FUNCTION "FC14 - AUTOMATIC" : VOID	// FC 14
VERSION : 0.1
BEGIN
// (block stored without names or comments; labels and parameter names are numbered)
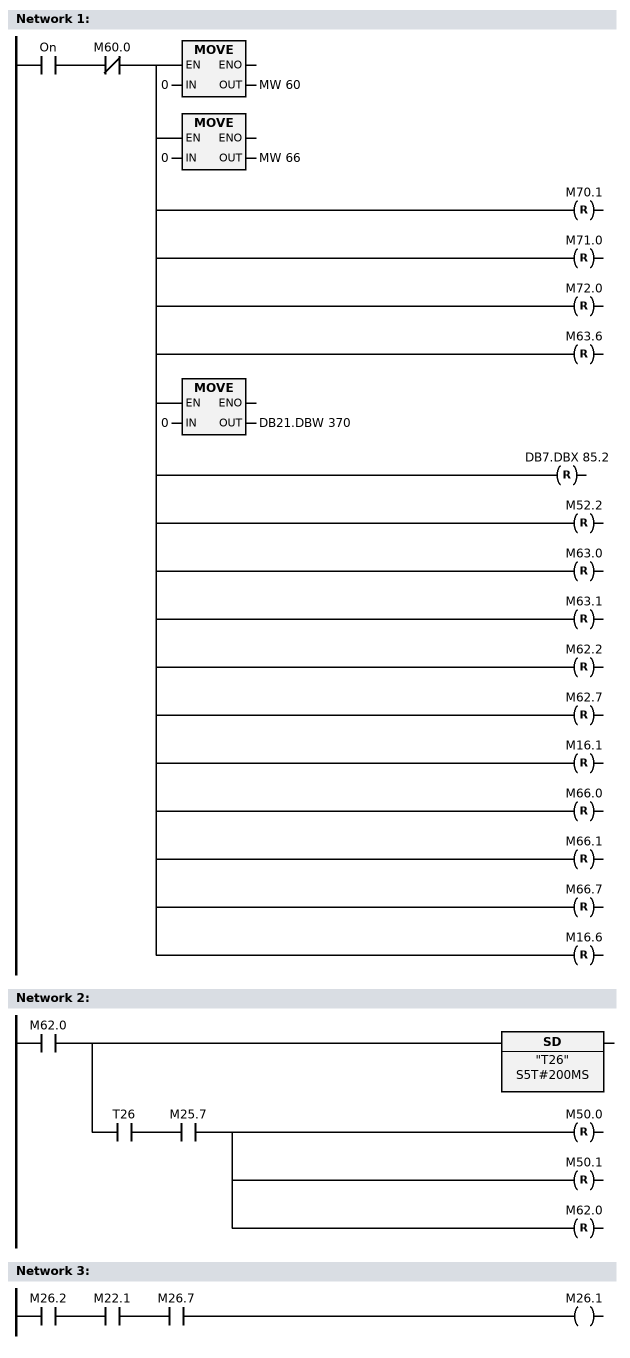
NETWORK
TITLE =
      A     "On";
      AN    "M60.0";
      =     L 24.0;
      A     L 24.0;
      JNB   M001;
      L     0;
      T     MW 60;
M001: NOP   0;
      A     L 24.0;
      JNB   M002;
      L     0;
      T     MW 66;
M002: NOP   0;
      A     L 24.0;
      BLD   102;
      R     "M70.1";
      A     L 24.0;
      BLD   102;
      R     "M71.0";
      A     L 24.0;
      BLD   102;
      R     "M72.0";
      A     L 24.0;
      BLD   102;
      R     "M63.6";
      A     L 24.0;
      JNB   M003;
      L     0;
      T     DB21.DBW 370;
M003: NOP   0;
      A     L 24.0;
      BLD   102;
      R     DB7.DBX 85.2;
      A     L 24.0;
      BLD   102;
      R     "M52.2";
      A     L 24.0;
      BLD   102;
      R     "M63.0";
      A     L 24.0;
      BLD   102;
      R     "M63.1";
      A     L 24.0;
      BLD   102;
      R     "M62.2";
      A     L 24.0;
      BLD   102;
      R     "M62.7";
      A     L 24.0;
      BLD   102;
      R     "M16.1";
      A     L 24.0;
      BLD   102;
      R     "M66.0";
      A     L 24.0;
      BLD   102;
      R     "M66.1";
      A     L 24.0;
      BLD   102;
      R     "M66.7";
      A     L 24.0;
      BLD   102;
      R     "M16.6";
NETWORK
TITLE =
      A     "M62.0";
      =     L 24.0;
      A     L 24.0;
      BLD   102;
      L     S5T#200MS;
      SD    "T26";
      A     L 24.0;
      A     "T26";
      A     "M25.7";
      R     "M50.0";
      R     "M50.1";
      R     "M62.0";
NETWORK
TITLE =
      A     "M26.2";
      A     "M22.1";
      A     "M26.7";
      =     "M26.1";
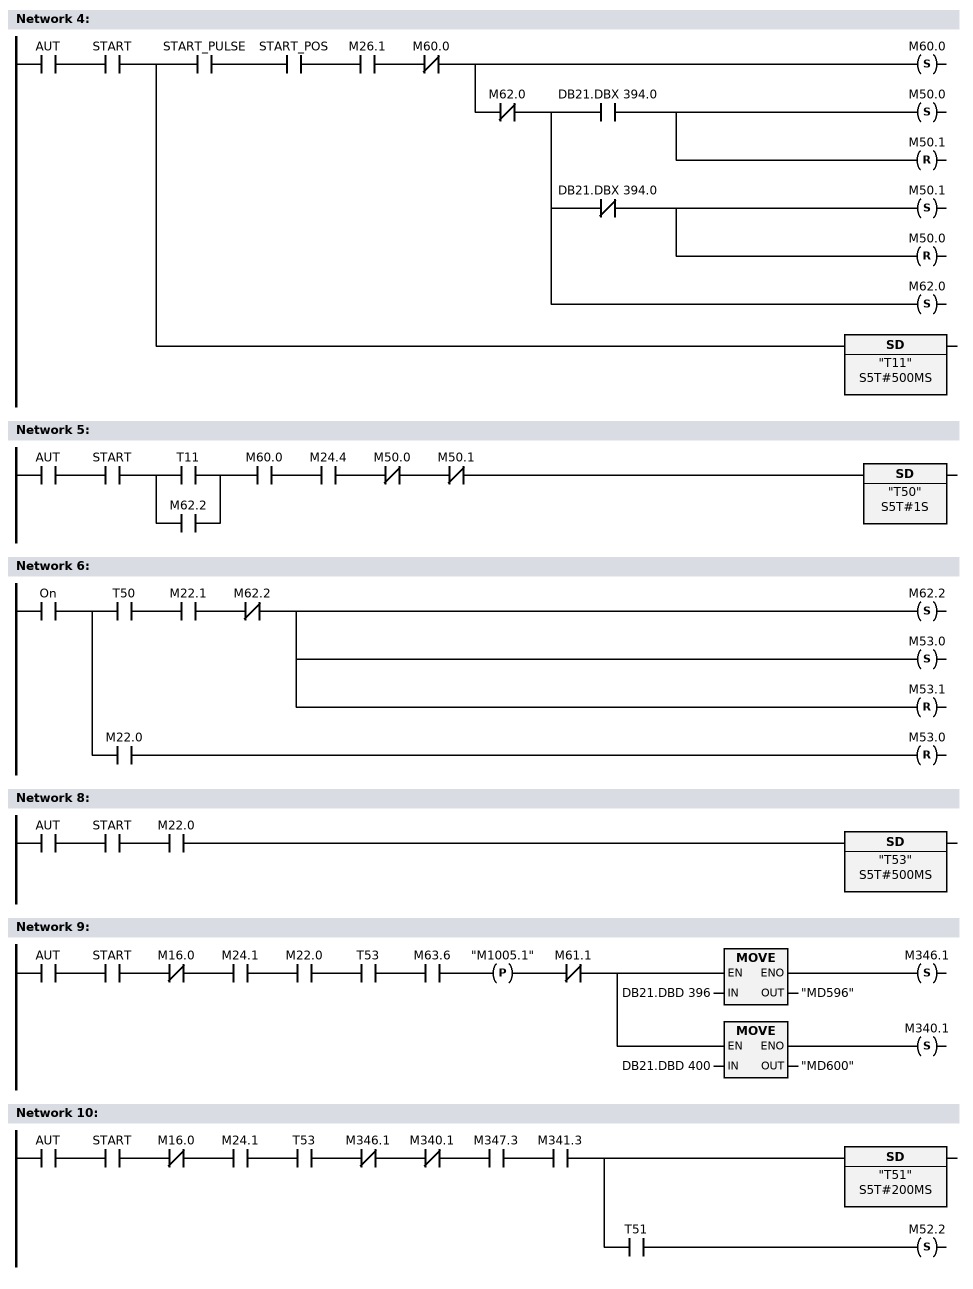
NETWORK
TITLE =
      A     "AUT";
      A     "START";
      =     L 24.0;
      A     L 24.0;
      A     "START_PULSE";
      A     "START_POS";
      A     "M26.1";
      AN    "M60.0";
      =     L 24.1;
      A     L 24.1;
      BLD   102;
      S     "M60.0";
      A     L 24.1;
      AN    "M62.0";
      =     L 24.2;
      A     L 24.2;
      A     DB21.DBX 394.0;
      S     "M50.0";
      R     "M50.1";
      A     L 24.2;
      AN    DB21.DBX 394.0;
      S     "M50.1";
      R     "M50.0";
      A     L 24.2;
      BLD   102;
      S     "M62.0";
      A     L 24.0;
      BLD   102;
      L     S5T#500MS;
      SD    "T11";
NETWORK
TITLE =
      A     "AUT";
      A     "START";
      A(;
      O     "T11";
      O     "M62.2";
      );
      A     "M60.0";
      A     "M24.4";
      AN    "M50.0";
      AN    "M50.1";
      L     S5T#1S;
      SD    "T50";
NETWORK
TITLE =
      A     "On";
      =     L 24.0;
      A     L 24.0;
      A     "T50";
      A     "M22.1";
      AN    "M62.2";
      S     "M62.2";
      S     "M53.0";
      R     "M53.1";
      A     L 24.0;
      A     "M22.0";
      R     "M53.0";
NETWORK
TITLE =
NETWORK
TITLE =
      A     "AUT";
      A     "START";
      A     "M22.0";
      L     S5T#500MS;
      SD    "T53";
NETWORK
TITLE =
      A     "AUT";
      A     "START";
      AN    "M16.0";
      A     "M24.1";
      A     "M22.0";
      A     "T53";
      A     "M63.6";
      FP    "M1005.1";
      AN    "M61.1";
      =     L 24.0;
      A     L 24.0;
      JNB   M004;
      L     DB21.DBD 396;
      T     "MD596";
      SET;
      SAVE;
      CLR;
M004: A     BR;
      S     "M346.1";
      A     L 24.0;
      JNB   M005;
      L     DB21.DBD 400;
      T     "MD600";
      SET;
      SAVE;
      CLR;
M005: A     BR;
      S     "M340.1";
NETWORK
TITLE =
      A     "AUT";
      A     "START";
      AN    "M16.0";
      A     "M24.1";
      A     "T53";
      AN    "M346.1";
      AN    "M340.1";
      A     "M347.3";
      A     "M341.3";
      =     L 24.0;
      A     L 24.0;
      BLD   102;
      L     S5T#200MS;
      SD    "T51";
      A     L 24.0;
      A     "T51";
      S     "M52.2";
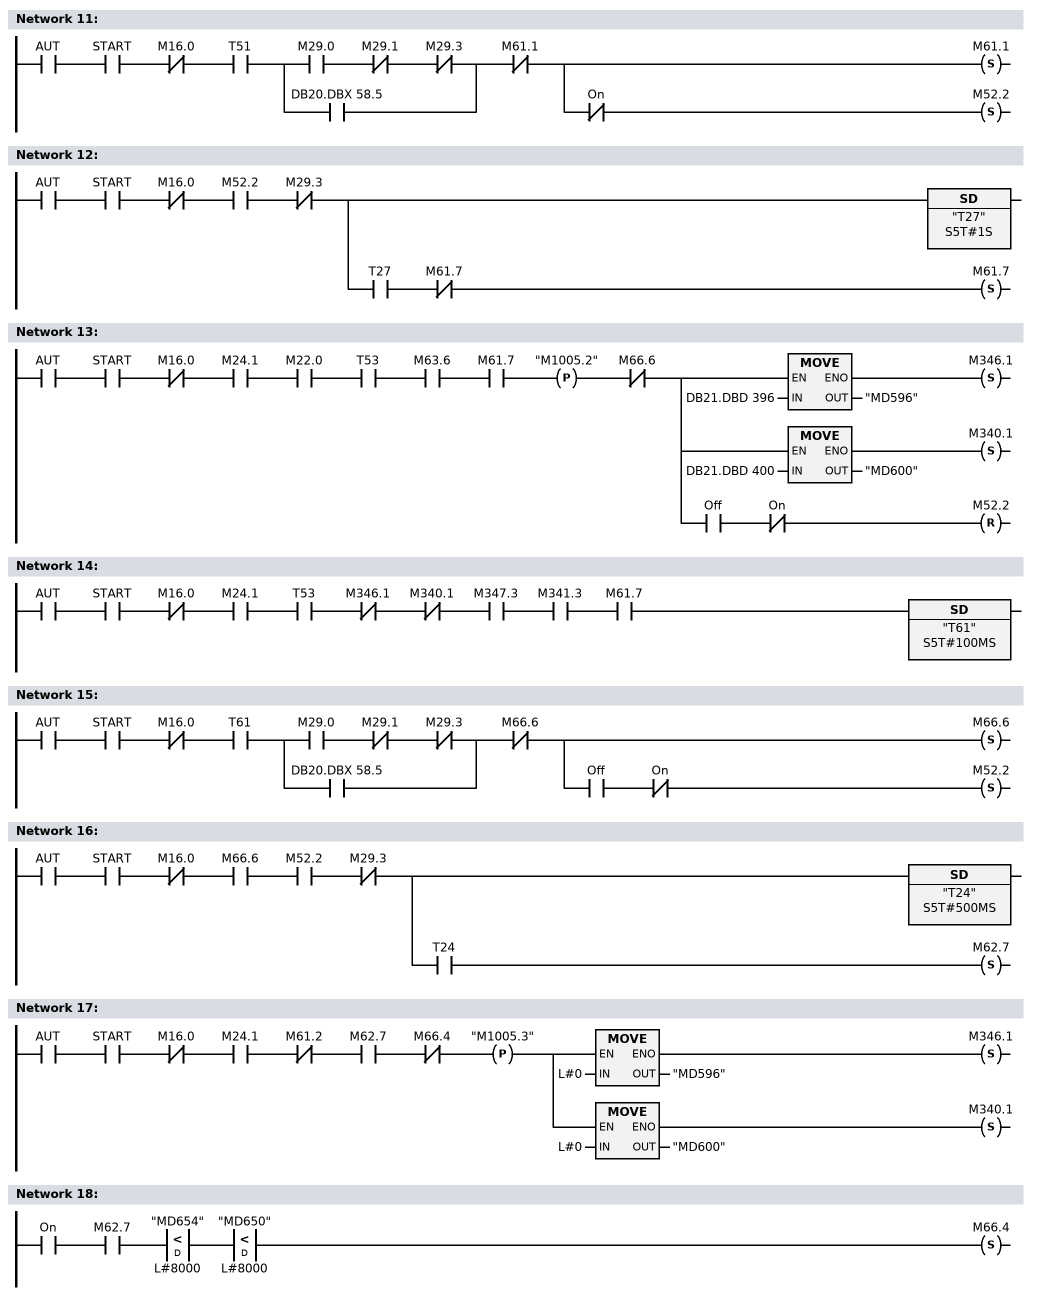
NETWORK
TITLE =
      A     "AUT";
      A     "START";
      AN    "M16.0";
      A     "T51";
      A(;
      A     "M29.0";
      AN    "M29.1";
      AN    "M29.3";
      O     DB20.DBX 58.5;
      );
      AN    "M61.1";
      =     L 24.0;
      A     L 24.0;
      BLD   102;
      S     "M61.1";
      A     L 24.0;
      AN    "On";
      S     "M52.2";
NETWORK
TITLE =
      A     "AUT";
      A     "START";
      AN    "M16.0";
      A     "M52.2";
      AN    "M29.3";
      =     L 24.0;
      A     L 24.0;
      BLD   102;
      L     S5T#1S;
      SD    "T27";
      A     L 24.0;
      A     "T27";
      AN    "M61.7";
      S     "M61.7";
NETWORK
TITLE =
      A     "AUT";
      A     "START";
      AN    "M16.0";
      A     "M24.1";
      A     "M22.0";
      A     "T53";
      A     "M63.6";
      A     "M61.7";
      FP    "M1005.2";
      AN    "M66.6";
      =     L 24.0;
      A     L 24.0;
      JNB   M006;
      L     DB21.DBD 396;
      T     "MD596";
      SET;
      SAVE;
      CLR;
M006: A     BR;
      S     "M346.1";
      A     L 24.0;
      JNB   M007;
      L     DB21.DBD 400;
      T     "MD600";
      SET;
      SAVE;
      CLR;
M007: A     BR;
      S     "M340.1";
      A     L 24.0;
      A     "Off";
      AN    "On";
      R     "M52.2";
NETWORK
TITLE =
      A     "AUT";
      A     "START";
      AN    "M16.0";
      A     "M24.1";
      A     "T53";
      AN    "M346.1";
      AN    "M340.1";
      A     "M347.3";
      A     "M341.3";
      A     "M61.7";
      L     S5T#100MS;
      SD    "T61";
NETWORK
TITLE =
      A     "AUT";
      A     "START";
      AN    "M16.0";
      A     "T61";
      A(;
      A     "M29.0";
      AN    "M29.1";
      AN    "M29.3";
      O     DB20.DBX 58.5;
      );
      AN    "M66.6";
      =     L 24.0;
      A     L 24.0;
      BLD   102;
      S     "M66.6";
      A     L 24.0;
      A     "Off";
      AN    "On";
      S     "M52.2";
NETWORK
TITLE =
      A     "AUT";
      A     "START";
      AN    "M16.0";
      A     "M66.6";
      A     "M52.2";
      AN    "M29.3";
      =     L 24.0;
      A     L 24.0;
      BLD   102;
      L     S5T#500MS;
      SD    "T24";
      A     L 24.0;
      A     "T24";
      S     "M62.7";
NETWORK
TITLE =
      A     "AUT";
      A     "START";
      AN    "M16.0";
      A     "M24.1";
      AN    "M61.2";
      A     "M62.7";
      AN    "M66.4";
      FP    "M1005.3";
      =     L 24.0;
      A     L 24.0;
      JNB   M008;
      L     L#0;
      T     "MD596";
      SET;
      SAVE;
      CLR;
M008: A     BR;
      S     "M346.1";
      A     L 24.0;
      JNB   M009;
      L     L#0;
      T     "MD600";
      SET;
      SAVE;
      CLR;
M009: A     BR;
      S     "M340.1";
NETWORK
TITLE =
      A     "On";
      A     "M62.7";
      A(;
      L     "MD654";
      L     L#8000;
      <D;
      );
      A(;
      L     "MD650";
      L     L#8000;
      <D;
      );
      S     "M66.4";
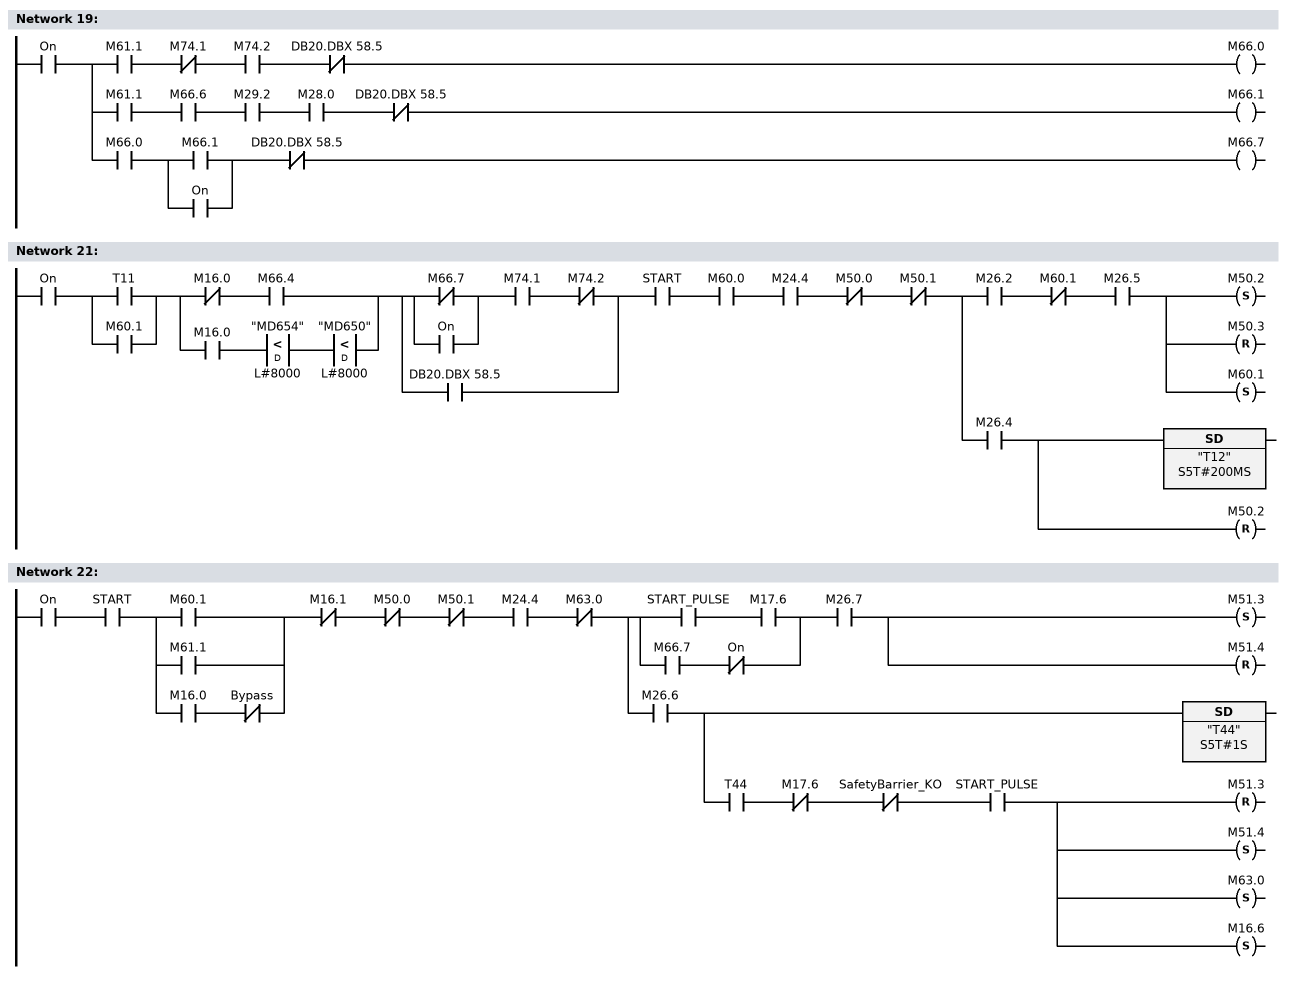
NETWORK
TITLE =
      A     "On";
      =     L 24.0;
      A     L 24.0;
      A     "M61.1";
      AN    "M74.1";
      A     "M74.2";
      AN    DB20.DBX 58.5;
      =     "M66.0";
      A     L 24.0;
      A     "M61.1";
      A     "M66.6";
      A     "M29.2";
      A     "M28.0";
      AN    DB20.DBX 58.5;
      =     "M66.1";
      A     L 24.0;
      A     "M66.0";
      A(;
      O     "M66.1";
      O     "On";
      );
      AN    DB20.DBX 58.5;
      =     "M66.7";
NETWORK
TITLE =
NETWORK
TITLE =
      A     "On";
      A(;
      O     "T11";
      O     "M60.1";
      );
      A(;
      AN    "M16.0";
      A     "M66.4";
      O;
      A     "M16.0";
      A(;
      L     "MD654";
      L     L#8000;
      <D;
      );
      A(;
      L     "MD650";
      L     L#8000;
      <D;
      );
      );
      A(;
      A(;
      ON    "M66.7";
      O     "On";
      );
      A     "M74.1";
      AN    "M74.2";
      O     DB20.DBX 58.5;
      );
      A     "START";
      A     "M60.0";
      A     "M24.4";
      AN    "M50.0";
      AN    "M50.1";
      =     L 24.0;
      A     L 24.0;
      A     "M26.2";
      AN    "M60.1";
      A     "M26.5";
      S     "M50.2";
      R     "M50.3";
      S     "M60.1";
      A     L 24.0;
      A     "M26.4";
      L     S5T#200MS;
      SD    "T12";
      R     "M50.2";
NETWORK
TITLE =
      A     "On";
      A     "START";
      A(;
      O     "M60.1";
      O     "M61.1";
      O;
      A     "M16.0";
      AN    "Bypass";
      );
      AN    "M16.1";
      AN    "M50.0";
      AN    "M50.1";
      A     "M24.4";
      AN    "M63.0";
      =     L 24.0;
      A     L 24.0;
      A(;
      A     "START_PULSE";
      A     "M17.6";
      O;
      A     "M66.7";
      AN    "On";
      );
      A     "M26.7";
      S     "M51.3";
      R     "M51.4";
      A     L 24.0;
      A     "M26.6";
      =     L 24.1;
      A     L 24.1;
      BLD   102;
      L     S5T#1S;
      SD    "T44";
      A     L 24.1;
      A     "T44";
      AN    "M17.6";
      AN    "SafetyBarrier_KO";
      A     "START_PULSE";
      R     "M51.3";
      S     "M51.4";
      S     "M63.0";
      S     "M16.6";
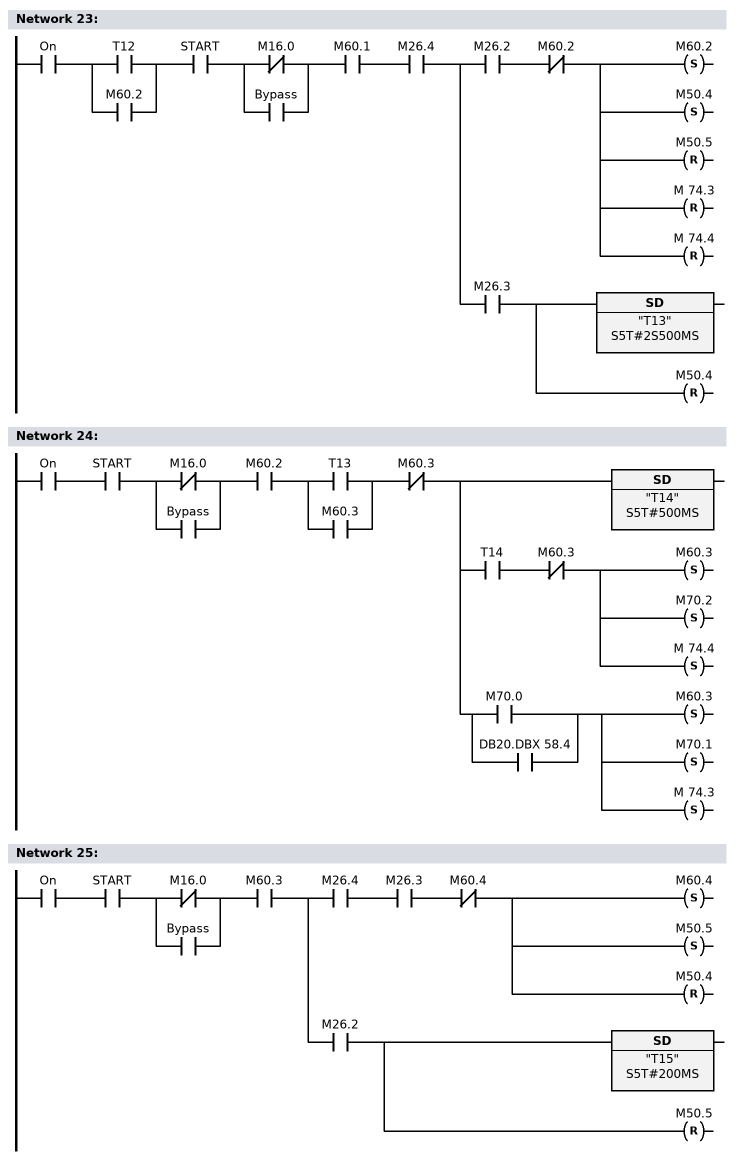
NETWORK
TITLE =
      A     "On";
      A(;
      O     "T12";
      O     "M60.2";
      );
      A     "START";
      A(;
      ON    "M16.0";
      O     "Bypass";
      );
      A     "M60.1";
      A     "M26.4";
      =     L 24.0;
      A     L 24.0;
      A     "M26.2";
      AN    "M60.2";
      S     "M60.2";
      S     "M50.4";
      R     "M50.5";
      R     M 74.3;
      R     M 74.4;
      A     L 24.0;
      A     "M26.3";
      L     S5T#2S500MS;
      SD    "T13";
      R     "M50.4";
NETWORK
TITLE =
      A     "On";
      A     "START";
      A(;
      ON    "M16.0";
      O     "Bypass";
      );
      A     "M60.2";
      A(;
      O     "T13";
      O     "M60.3";
      );
      AN    "M60.3";
      =     L 24.0;
      A     L 24.0;
      BLD   102;
      L     S5T#500MS;
      SD    "T14";
      A     L 24.0;
      A     "T14";
      AN    "M60.3";
      S     "M60.3";
      S     "M70.2";
      S     M 74.4;
      A     L 24.0;
      A(;
      O     "M70.0";
      O     DB20.DBX 58.4;
      );
      S     "M60.3";
      S     "M70.1";
      S     M 74.3;
NETWORK
TITLE =
      A     "On";
      A     "START";
      A(;
      ON    "M16.0";
      O     "Bypass";
      );
      A     "M60.3";
      =     L 24.0;
      A     L 24.0;
      A     "M26.4";
      A     "M26.3";
      AN    "M60.4";
      S     "M60.4";
      S     "M50.5";
      R     "M50.4";
      A     L 24.0;
      A     "M26.2";
      L     S5T#200MS;
      SD    "T15";
      R     "M50.5";
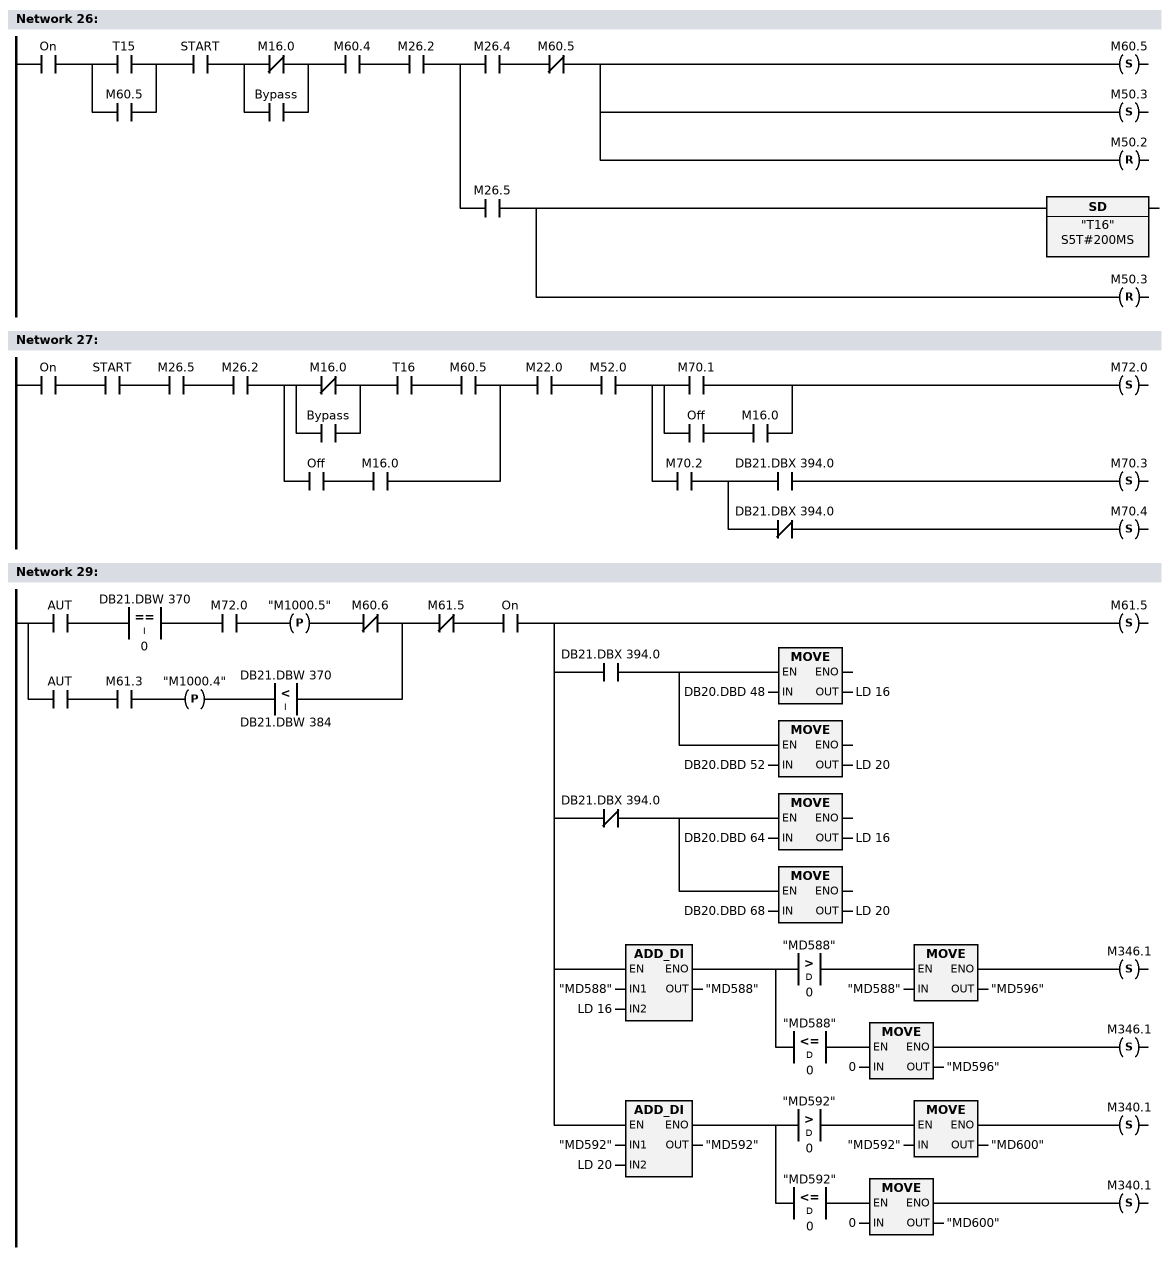
NETWORK
TITLE =
      A     "On";
      A(;
      O     "T15";
      O     "M60.5";
      );
      A     "START";
      A(;
      ON    "M16.0";
      O     "Bypass";
      );
      A     "M60.4";
      A     "M26.2";
      =     L 24.0;
      A     L 24.0;
      A     "M26.4";
      AN    "M60.5";
      S     "M60.5";
      S     "M50.3";
      R     "M50.2";
      A     L 24.0;
      A     "M26.5";
      L     S5T#200MS;
      SD    "T16";
      R     "M50.3";
NETWORK
TITLE =
      A     "On";
      A     "START";
      A     "M26.5";
      A     "M26.2";
      A(;
      A(;
      ON    "M16.0";
      O     "Bypass";
      );
      A     "T16";
      A     "M60.5";
      O;
      A     "Off";
      A     "M16.0";
      );
      A     "M22.0";
      A     "M52.0";
      =     L 24.0;
      A     L 24.0;
      A(;
      O     "M70.1";
      O;
      A     "Off";
      A     "M16.0";
      );
      S     "M72.0";
      A     L 24.0;
      A     "M70.2";
      =     L 24.1;
      A     L 24.1;
      A     DB21.DBX 394.0;
      S     "M70.3";
      A     L 24.1;
      AN    DB21.DBX 394.0;
      S     "M70.4";
NETWORK
TITLE =
NETWORK
TITLE =
      A(;
      A     "AUT";
      A(;
      L     DB21.DBW 370;
      L     0;
      ==I;
      );
      A     "M72.0";
      FP    "M1000.5";
      AN    "M60.6";
      O(;
      A     "AUT";
      A     "M61.3";
      FP    "M1000.4";
      A(;
      L     DB21.DBW 370;
      L     DB21.DBW 384;
      <I;
      );
      );
      );
      AN    "M61.5";
      A     "On";
      =     L 24.0;
      A     L 24.0;
      BLD   102;
      S     "M61.5";
      A     L 24.0;
      A     DB21.DBX 394.0;
      =     L 24.1;
      A     L 24.1;
      JNB   M010;
      L     DB20.DBD 48;
      T     LD 16;
M010: NOP   0;
      A     L 24.1;
      JNB   M011;
      L     DB20.DBD 52;
      T     LD 20;
M011: NOP   0;
      A     L 24.0;
      AN    DB21.DBX 394.0;
      =     L 24.1;
      A     L 24.1;
      JNB   M012;
      L     DB20.DBD 64;
      T     LD 16;
M012: NOP   0;
      A     L 24.1;
      JNB   M013;
      L     DB20.DBD 68;
      T     LD 20;
M013: NOP   0;
      A     L 24.0;
      JNB   M014;
      L     "MD588";
      L     LD 16;
      +D;
      T     "MD588";
      AN    OV;
      SAVE;
      CLR;
M014: A     BR;
      =     L 24.1;
      A     L 24.1;
      A(;
      L     "MD588";
      L     0;
      >D;
      );
      JNB   M015;
      L     "MD588";
      T     "MD596";
      SET;
      SAVE;
      CLR;
M015: A     BR;
      S     "M346.1";
      A     L 24.1;
      A(;
      L     "MD588";
      L     0;
      <=D;
      );
      JNB   M016;
      L     0;
      T     "MD596";
      SET;
      SAVE;
      CLR;
M016: A     BR;
      S     "M346.1";
      A     L 24.0;
      JNB   M017;
      L     "MD592";
      L     LD 20;
      +D;
      T     "MD592";
      AN    OV;
      SAVE;
      CLR;
M017: A     BR;
      =     L 24.1;
      A     L 24.1;
      A(;
      L     "MD592";
      L     0;
      >D;
      );
      JNB   M018;
      L     "MD592";
      T     "MD600";
      SET;
      SAVE;
      CLR;
M018: A     BR;
      S     "M340.1";
      A     L 24.1;
      A(;
      L     "MD592";
      L     0;
      <=D;
      );
      JNB   M019;
      L     0;
      T     "MD600";
      SET;
      SAVE;
      CLR;
M019: A     BR;
      S     "M340.1";
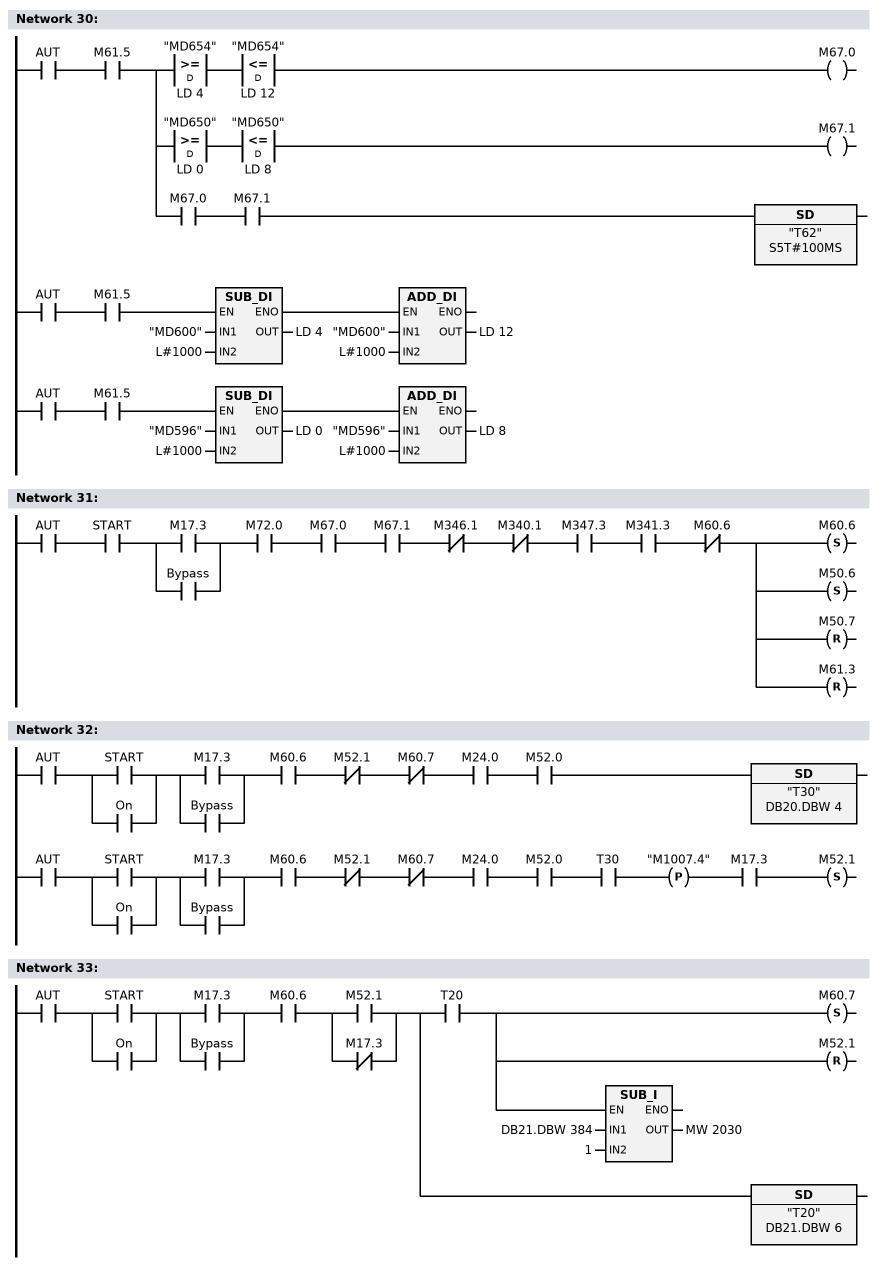
NETWORK
TITLE =
      A     "AUT";
      A     "M61.5";
      =     L 24.0;
      A(;
      A     L 24.0;
      JNB   M020;
      L     "MD600";
      L     L#1000;
      -D;
      T     LD 4;
      AN    OV;
      SAVE;
      CLR;
M020: A     BR;
      );
      JNB   M021;
      L     "MD600";
      L     L#1000;
      +D;
      T     LD 12;
M021: NOP   0;
      A(;
      A     L 24.0;
      JNB   M022;
      L     "MD596";
      L     L#1000;
      -D;
      T     LD 0;
      AN    OV;
      SAVE;
      CLR;
M022: A     BR;
      );
      JNB   M023;
      L     "MD596";
      L     L#1000;
      +D;
      T     LD 8;
M023: NOP   0;
      A     L 24.0;
      A(;
      L     "MD654";
      L     LD 4;
      >=D;
      );
      A(;
      L     "MD654";
      L     LD 12;
      <=D;
      );
      =     "M67.0";
      A     L 24.0;
      A(;
      L     "MD650";
      L     LD 0;
      >=D;
      );
      A(;
      L     "MD650";
      L     LD 8;
      <=D;
      );
      =     "M67.1";
      A     L 24.0;
      A     "M67.0";
      A     "M67.1";
      L     S5T#100MS;
      SD    "T62";
NETWORK
TITLE =
      A     "AUT";
      A     "START";
      A(;
      O     "M17.3";
      O     "Bypass";
      );
      A     "M72.0";
      A     "M67.0";
      A     "M67.1";
      AN    "M346.1";
      AN    "M340.1";
      A     "M347.3";
      A     "M341.3";
      AN    "M60.6";
      S     "M60.6";
      S     "M50.6";
      R     "M50.7";
      R     "M61.3";
NETWORK
TITLE =
      A     "AUT";
      A(;
      O     "START";
      O     "On";
      );
      A(;
      O     "M17.3";
      O     "Bypass";
      );
      A     "M60.6";
      AN    "M52.1";
      AN    "M60.7";
      A     "M24.0";
      A     "M52.0";
      =     L 24.0;
      A     L 24.0;
      BLD   102;
      L     DB20.DBW 4;
      SD    "T30";
      A(;
      A     L 24.0;
      A     "T30";
      FP    "M1007.4";
      );
      A     "M17.3";
      S     "M52.1";
NETWORK
TITLE =
      A     "AUT";
      A(;
      O     "START";
      O     "On";
      );
      A(;
      O     "M17.3";
      O     "Bypass";
      );
      A     "M60.6";
      A(;
      O     "M52.1";
      ON    "M17.3";
      );
      =     L 24.0;
      A     L 24.0;
      A     "T20";
      =     L 24.1;
      A     L 24.1;
      BLD   102;
      S     "M60.7";
      A     L 24.1;
      BLD   102;
      R     "M52.1";
      A     L 24.1;
      JNB   M024;
      L     DB21.DBW 384;
      L     1;
      -I;
      T     MW 2030;
M024: NOP   0;
      A     L 24.0;
      BLD   102;
      L     DB21.DBW 6;
      SD    "T20";
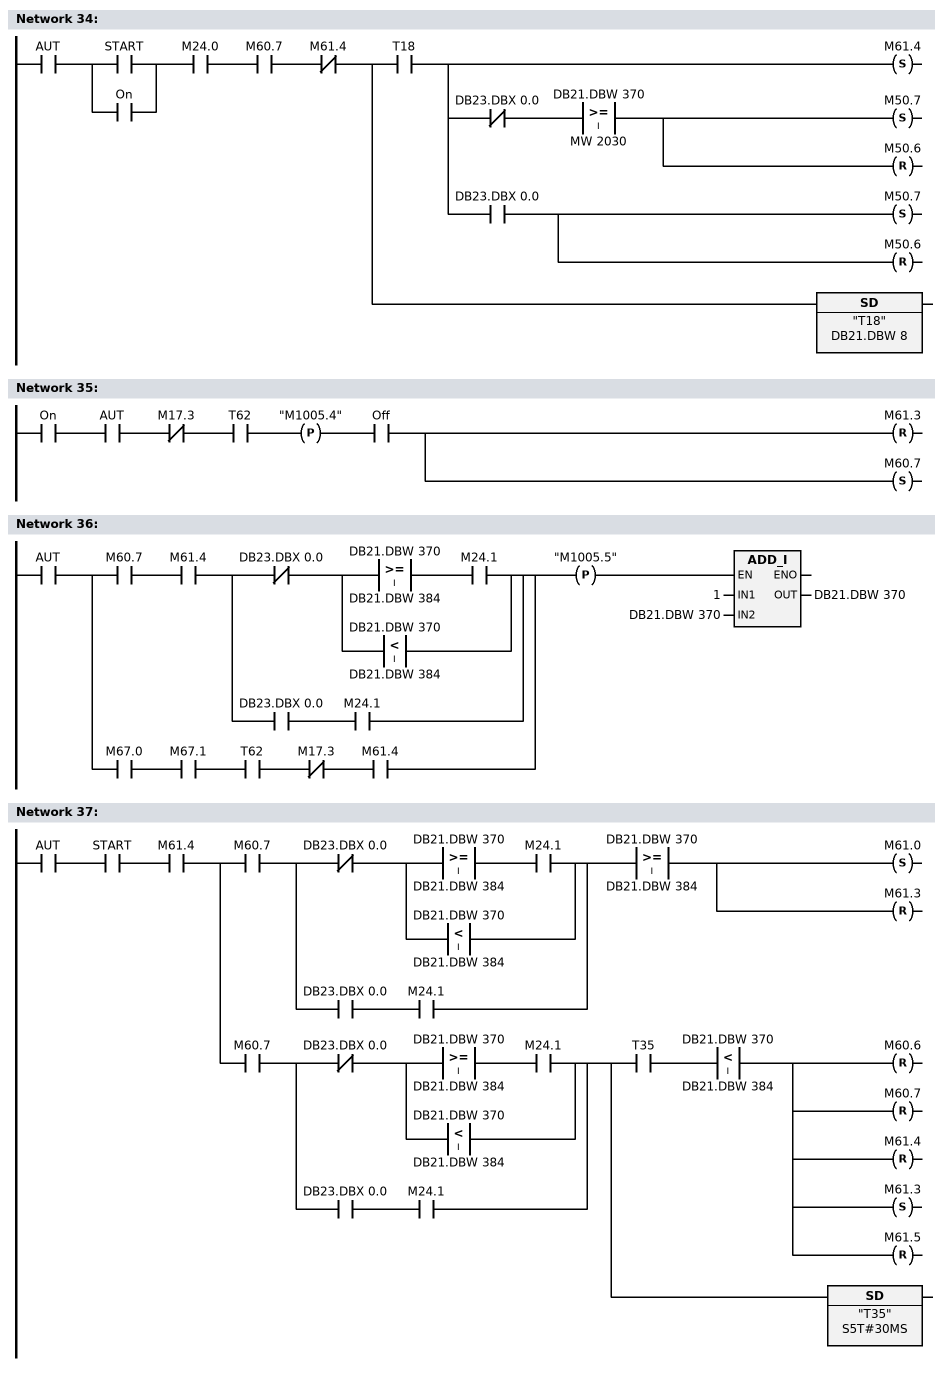
NETWORK
TITLE =
      A     "AUT";
      A(;
      O     "START";
      O     "On";
      );
      A     "M24.0";
      A     "M60.7";
      AN    "M61.4";
      =     L 24.0;
      A     L 24.0;
      A     "T18";
      =     L 24.1;
      A     L 24.1;
      BLD   102;
      S     "M61.4";
      A     L 24.1;
      AN    DB23.DBX 0.0;
      A(;
      L     DB21.DBW 370;
      L     MW 2030;
      >=I;
      );
      S     "M50.7";
      R     "M50.6";
      A     L 24.1;
      A     DB23.DBX 0.0;
      S     "M50.7";
      R     "M50.6";
      A     L 24.0;
      BLD   102;
      L     DB21.DBW 8;
      SD    "T18";
NETWORK
TITLE =
      A     "On";
      A     "AUT";
      AN    "M17.3";
      A     "T62";
      FP    "M1005.4";
      A     "Off";
      R     "M61.3";
      S     "M60.7";
NETWORK
TITLE =
      A     "AUT";
      A(;
      A     "M60.7";
      A     "M61.4";
      A(;
      AN    DB23.DBX 0.0;
      A(;
      A(;
      L     DB21.DBW 370;
      L     DB21.DBW 384;
      >=I;
      );
      A     "M24.1";
      O(;
      L     DB21.DBW 370;
      L     DB21.DBW 384;
      <I;
      );
      );
      O;
      A     DB23.DBX 0.0;
      A     "M24.1";
      );
      O;
      A     "M67.0";
      A     "M67.1";
      A     "T62";
      AN    "M17.3";
      A     "M61.4";
      );
      FP    "M1005.5";
      JNB   M025;
      L     1;
      L     DB21.DBW 370;
      +I;
      T     DB21.DBW 370;
M025: NOP   0;
NETWORK
TITLE =
      A     "AUT";
      A     "START";
      A     "M61.4";
      =     L 24.0;
      A     L 24.0;
      A     "M60.7";
      A(;
      AN    DB23.DBX 0.0;
      A(;
      A(;
      L     DB21.DBW 370;
      L     DB21.DBW 384;
      >=I;
      );
      A     "M24.1";
      O(;
      L     DB21.DBW 370;
      L     DB21.DBW 384;
      <I;
      );
      );
      O;
      A     DB23.DBX 0.0;
      A     "M24.1";
      );
      A(;
      L     DB21.DBW 370;
      L     DB21.DBW 384;
      >=I;
      );
      S     "M61.0";
      R     "M61.3";
      A     L 24.0;
      A     "M60.7";
      A(;
      AN    DB23.DBX 0.0;
      A(;
      A(;
      L     DB21.DBW 370;
      L     DB21.DBW 384;
      >=I;
      );
      A     "M24.1";
      O(;
      L     DB21.DBW 370;
      L     DB21.DBW 384;
      <I;
      );
      );
      O;
      A     DB23.DBX 0.0;
      A     "M24.1";
      );
      =     L 24.1;
      A     L 24.1;
      A     "T35";
      A(;
      L     DB21.DBW 370;
      L     DB21.DBW 384;
      <I;
      );
      R     "M60.6";
      R     "M60.7";
      R     "M61.4";
      S     "M61.3";
      R     "M61.5";
      A     L 24.1;
      BLD   102;
      L     S5T#30MS;
      SD    "T35";
NETWORK
TITLE =
NETWORK
TITLE =
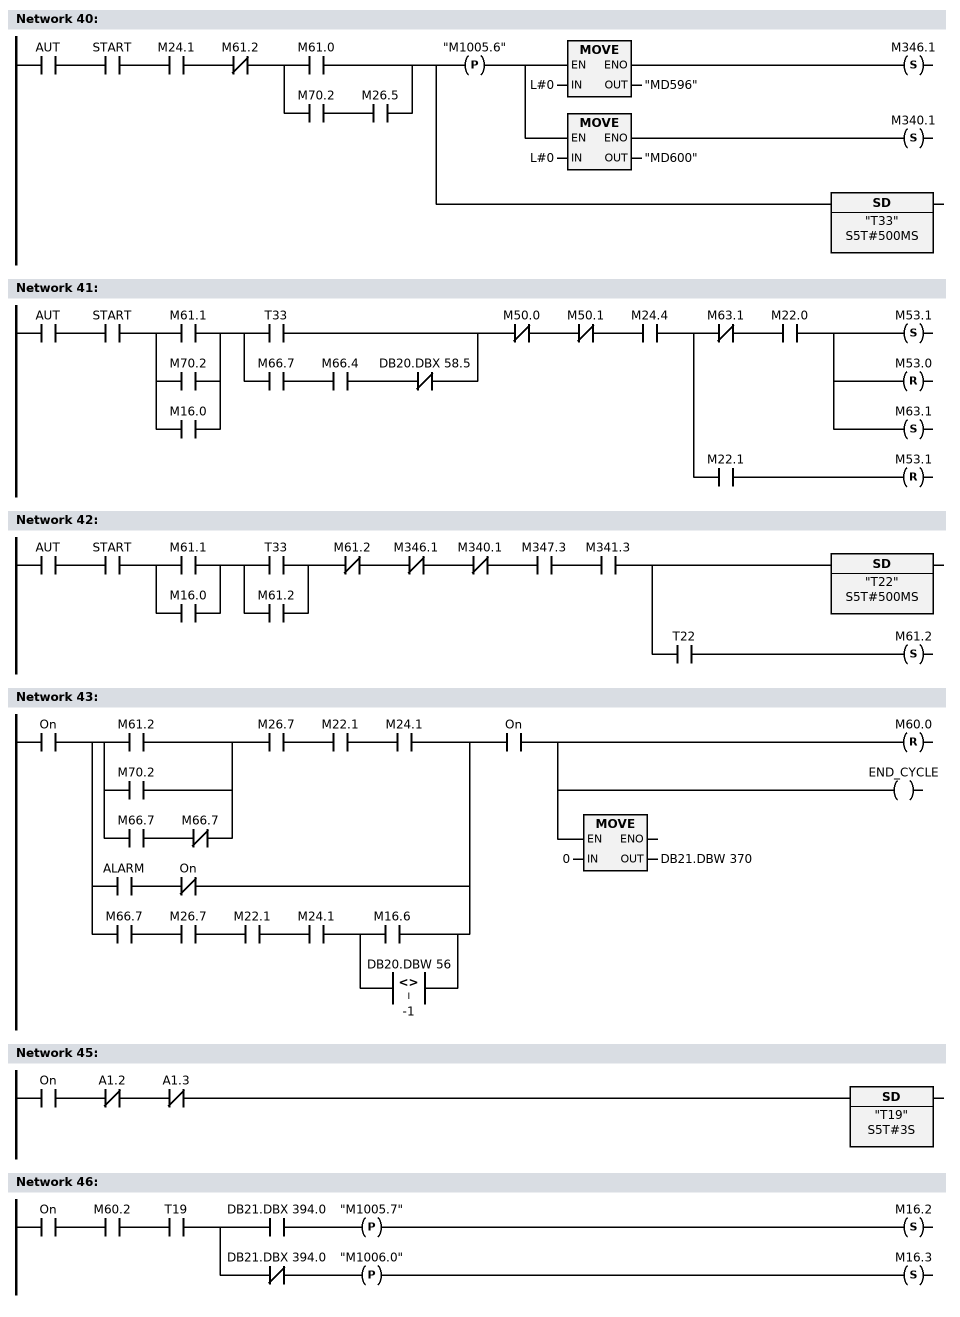
NETWORK
TITLE =
      A     "AUT";
      A     "START";
      A     "M24.1";
      AN    "M61.2";
      A(;
      O     "M61.0";
      O;
      A     "M70.2";
      A     "M26.5";
      );
      =     L 24.0;
      A     L 24.0;
      FP    "M1005.6";
      =     L 24.1;
      A     L 24.1;
      JNB   M026;
      L     L#0;
      T     "MD596";
      SET;
      SAVE;
      CLR;
M026: A     BR;
      S     "M346.1";
      A     L 24.1;
      JNB   M027;
      L     L#0;
      T     "MD600";
      SET;
      SAVE;
      CLR;
M027: A     BR;
      S     "M340.1";
      A     L 24.0;
      BLD   102;
      L     S5T#500MS;
      SD    "T33";
NETWORK
TITLE =
      A     "AUT";
      A     "START";
      A(;
      O     "M61.1";
      O     "M70.2";
      O     "M16.0";
      );
      A(;
      O     "T33";
      O;
      A     "M66.7";
      A     "M66.4";
      AN    DB20.DBX 58.5;
      );
      AN    "M50.0";
      AN    "M50.1";
      A     "M24.4";
      =     L 24.0;
      A     L 24.0;
      AN    "M63.1";
      A     "M22.0";
      S     "M53.1";
      R     "M53.0";
      S     "M63.1";
      A     L 24.0;
      A     "M22.1";
      R     "M53.1";
NETWORK
TITLE =
      A     "AUT";
      A     "START";
      A(;
      O     "M61.1";
      O     "M16.0";
      );
      A(;
      O     "T33";
      O     "M61.2";
      );
      AN    "M61.2";
      AN    "M346.1";
      AN    "M340.1";
      A     "M347.3";
      A     "M341.3";
      =     L 24.0;
      A     L 24.0;
      BLD   102;
      L     S5T#500MS;
      SD    "T22";
      A     L 24.0;
      A     "T22";
      S     "M61.2";
NETWORK
TITLE =
      A     "On";
      A(;
      A(;
      O     "M61.2";
      O     "M70.2";
      O;
      A     "M66.7";
      AN    "M66.7";
      );
      A     "M26.7";
      A     "M22.1";
      A     "M24.1";
      O;
      A     "ALARM";
      AN    "On";
      O;
      A     "M66.7";
      A     "M26.7";
      A     "M22.1";
      A     "M24.1";
      A(;
      O     "M16.6";
      O(;
      L     DB20.DBW 56;
      L     -1;
      <>I;
      );
      );
      );
      A     "On";
      =     L 24.0;
      A     L 24.0;
      BLD   102;
      R     "M60.0";
      A     L 24.0;
      BLD   102;
      =     "END_CYCLE";
      A     L 24.0;
      JNB   M028;
      L     0;
      T     DB21.DBW 370;
M028: NOP   0;
NETWORK
TITLE =
NETWORK
TITLE =
      A     "On";
      AN    "A1.2";
      AN    "A1.3";
      L     S5T#3S;
      SD    "T19";
NETWORK
TITLE =
      A     "On";
      A     "M60.2";
      A     "T19";
      =     L 24.0;
      A     L 24.0;
      A     DB21.DBX 394.0;
      FP    "M1005.7";
      S     "M16.2";
      A     L 24.0;
      AN    DB21.DBX 394.0;
      FP    "M1006.0";
      S     "M16.3";
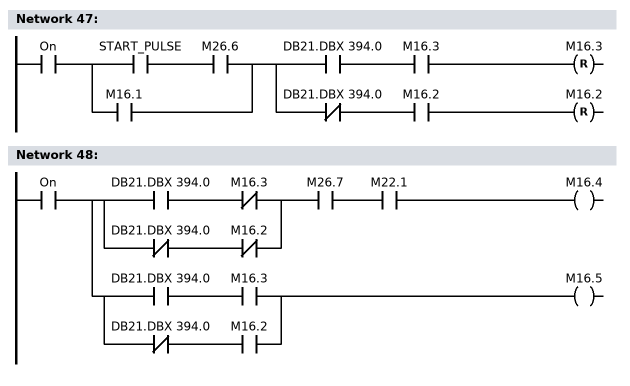
NETWORK
TITLE =
      A     "On";
      A(;
      A     "START_PULSE";
      A     "M26.6";
      O     "M16.1";
      );
      =     L 24.0;
      A     L 24.0;
      A     DB21.DBX 394.0;
      A     "M16.3";
      R     "M16.3";
      A     L 24.0;
      AN    DB21.DBX 394.0;
      A     "M16.2";
      R     "M16.2";
NETWORK
TITLE =
      A     "On";
      =     L 24.0;
      A     L 24.0;
      A(;
      A     DB21.DBX 394.0;
      AN    "M16.3";
      O;
      AN    DB21.DBX 394.0;
      AN    "M16.2";
      );
      A     "M26.7";
      A     "M22.1";
      =     "M16.4";
      A     L 24.0;
      A(;
      A     DB21.DBX 394.0;
      A     "M16.3";
      O;
      AN    DB21.DBX 394.0;
      A     "M16.2";
      );
      =     "M16.5";
END_FUNCTION

FUNCTION "FC16 - ALARMS" : VOID	// FC 16
VERSION : 0.1
BEGIN
// (block stored without names or comments; labels and parameter names are numbered)
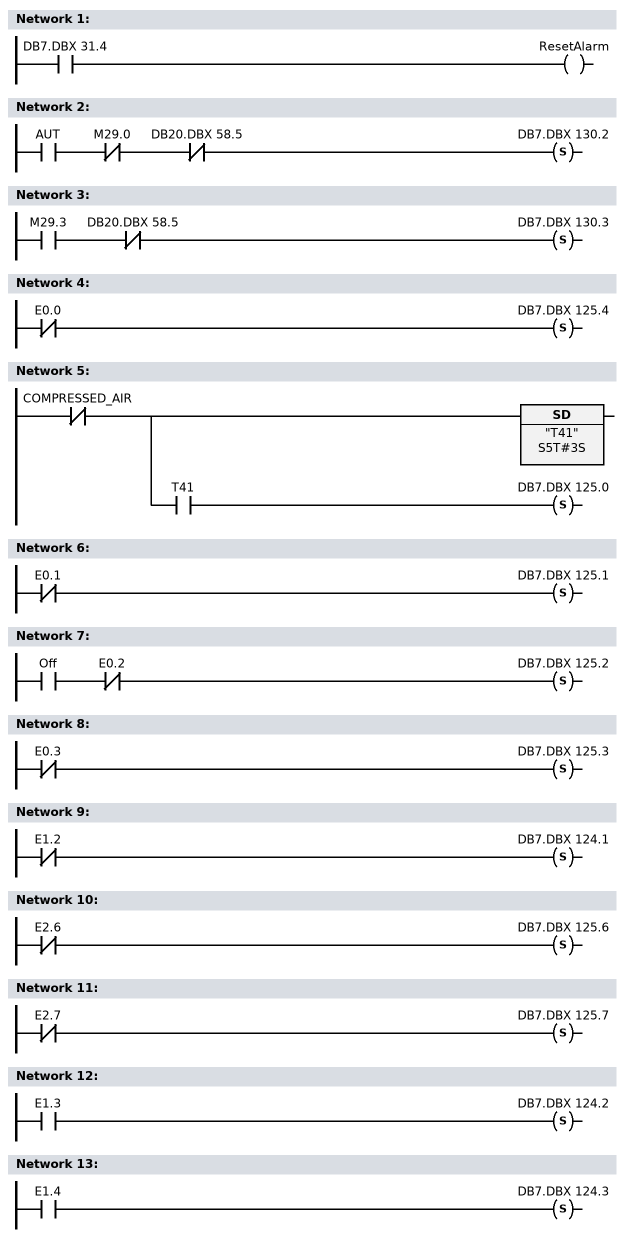
NETWORK
TITLE =
      A     DB7.DBX 31.4;
      =     "ResetAlarm";
NETWORK
TITLE =
      A     "AUT";
      AN    "M29.0";
      AN    DB20.DBX 58.5;
      S     DB7.DBX 130.2;
NETWORK
TITLE =
      A     "M29.3";
      AN    DB20.DBX 58.5;
      S     DB7.DBX 130.3;
NETWORK
TITLE =
      AN    "E0.0";
      S     DB7.DBX 125.4;
NETWORK
TITLE =
      AN    "COMPRESSED_AIR";
      =     L 1.0;
      A     L 1.0;
      BLD   102;
      L     S5T#3S;
      SD    "T41";
      A     L 1.0;
      A     "T41";
      S     DB7.DBX 125.0;
NETWORK
TITLE =
      AN    "E0.1";
      S     DB7.DBX 125.1;
NETWORK
TITLE =
      A     "Off";
      AN    "E0.2";
      S     DB7.DBX 125.2;
NETWORK
TITLE =
      AN    "E0.3";
      S     DB7.DBX 125.3;
NETWORK
TITLE =
      AN    "E1.2";
      S     DB7.DBX 124.1;
NETWORK
TITLE =
      AN    "E2.6";
      S     DB7.DBX 125.6;
NETWORK
TITLE =
      AN    "E2.7";
      S     DB7.DBX 125.7;
NETWORK
TITLE =
      A     "E1.3";
      S     DB7.DBX 124.2;
NETWORK
TITLE =
      A     "E1.4";
      S     DB7.DBX 124.3;
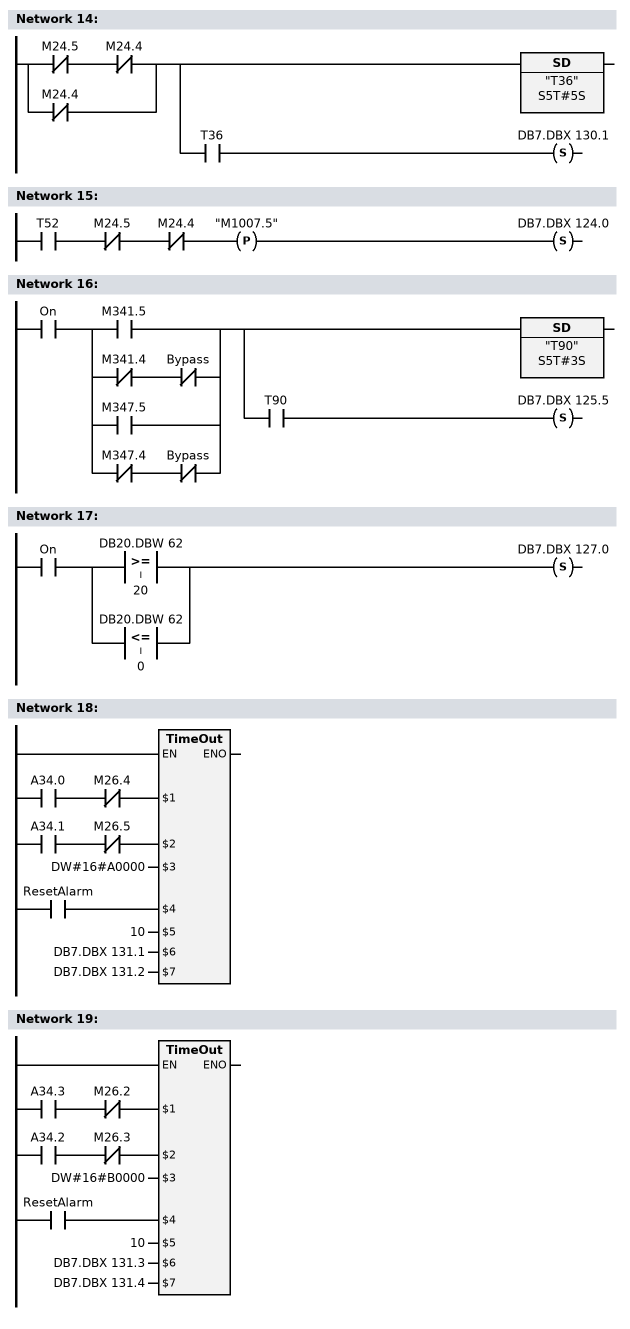
NETWORK
TITLE =
      AN    "M24.5";
      AN    "M24.4";
      ON    "M24.4";
      =     L 1.0;
      A     L 1.0;
      BLD   102;
      L     S5T#5S;
      SD    "T36";
      A     L 1.0;
      A     "T36";
      S     DB7.DBX 130.1;
NETWORK
TITLE =
      A     "T52";
      AN    "M24.5";
      AN    "M24.4";
      FP    "M1007.5";
      S     DB7.DBX 124.0;
NETWORK
TITLE =
      A     "On";
      A(;
      O     "M341.5";
      O;
      AN    "M341.4";
      AN    "Bypass";
      O     "M347.5";
      O;
      AN    "M347.4";
      AN    "Bypass";
      );
      =     L 1.0;
      A     L 1.0;
      BLD   102;
      L     S5T#3S;
      SD    "T90";
      A     L 1.0;
      A     "T90";
      S     DB7.DBX 125.5;
NETWORK
TITLE =
      A     "On";
      A(;
      O(;
      L     DB20.DBW 62;
      L     20;
      >=I;
      );
      O(;
      L     DB20.DBW 62;
      L     0;
      <=I;
      );
      );
      S     DB7.DBX 127.0;
NETWORK
TITLE =
      A     "A34.0";
      AN    "M26.4";
      =     L 1.0;
      BLD   103;
      A     "A34.1";
      AN    "M26.5";
      =     L 1.1;
      BLD   103;
      A     "ResetAlarm";
      =     L 1.2;
      BLD   103;
      CALL  "TimeOut" (
           $1                       := L 1.0,
           $2                       := L 1.1,
           $3                       := DW#16#A0000,
           $4                       := L 1.2,
           $5                       := 10,
           $6                       := DB7.DBX 131.1,
           $7                       := DB7.DBX 131.2);
      NOP   0;
NETWORK
TITLE =
      A     "A34.3";
      AN    "M26.2";
      =     L 1.0;
      BLD   103;
      A     "A34.2";
      AN    "M26.3";
      =     L 1.1;
      BLD   103;
      A     "ResetAlarm";
      =     L 1.2;
      BLD   103;
      CALL  "TimeOut" (
           $1                       := L 1.0,
           $2                       := L 1.1,
           $3                       := DW#16#B0000,
           $4                       := L 1.2,
           $5                       := 10,
           $6                       := DB7.DBX 131.3,
           $7                       := DB7.DBX 131.4);
      NOP   0;
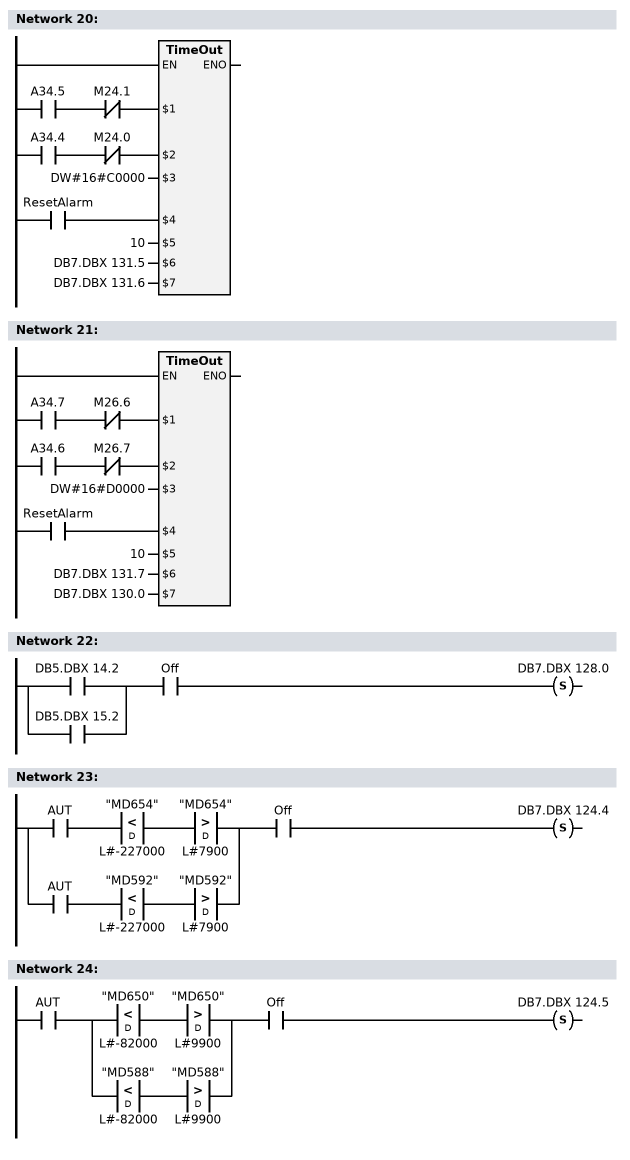
NETWORK
TITLE =
      A     "A34.5";
      AN    "M24.1";
      =     L 1.0;
      BLD   103;
      A     "A34.4";
      AN    "M24.0";
      =     L 1.1;
      BLD   103;
      A     "ResetAlarm";
      =     L 1.2;
      BLD   103;
      CALL  "TimeOut" (
           $1                       := L 1.0,
           $2                       := L 1.1,
           $3                       := DW#16#C0000,
           $4                       := L 1.2,
           $5                       := 10,
           $6                       := DB7.DBX 131.5,
           $7                       := DB7.DBX 131.6);
      NOP   0;
NETWORK
TITLE =
      A     "A34.7";
      AN    "M26.6";
      =     L 1.0;
      BLD   103;
      A     "A34.6";
      AN    "M26.7";
      =     L 1.1;
      BLD   103;
      A     "ResetAlarm";
      =     L 1.2;
      BLD   103;
      CALL  "TimeOut" (
           $1                       := L 1.0,
           $2                       := L 1.1,
           $3                       := DW#16#D0000,
           $4                       := L 1.2,
           $5                       := 10,
           $6                       := DB7.DBX 131.7,
           $7                       := DB7.DBX 130.0);
      NOP   0;
NETWORK
TITLE =
      A(;
      O     DB5.DBX 14.2;
      O     DB5.DBX 15.2;
      );
      A     "Off";
      S     DB7.DBX 128.0;
NETWORK
TITLE =
      A(;
      A     "AUT";
      A(;
      L     "MD654";
      L     L#-227000;
      <D;
      );
      A(;
      L     "MD654";
      L     L#7900;
      >D;
      );
      O;
      A     "AUT";
      A(;
      L     "MD592";
      L     L#-227000;
      <D;
      );
      A(;
      L     "MD592";
      L     L#7900;
      >D;
      );
      );
      A     "Off";
      S     DB7.DBX 124.4;
NETWORK
TITLE =
      A     "AUT";
      A(;
      A(;
      L     "MD650";
      L     L#-82000;
      <D;
      );
      A(;
      L     "MD650";
      L     L#9900;
      >D;
      );
      O;
      A(;
      L     "MD588";
      L     L#-82000;
      <D;
      );
      A(;
      L     "MD588";
      L     L#9900;
      >D;
      );
      );
      A     "Off";
      S     DB7.DBX 124.5;
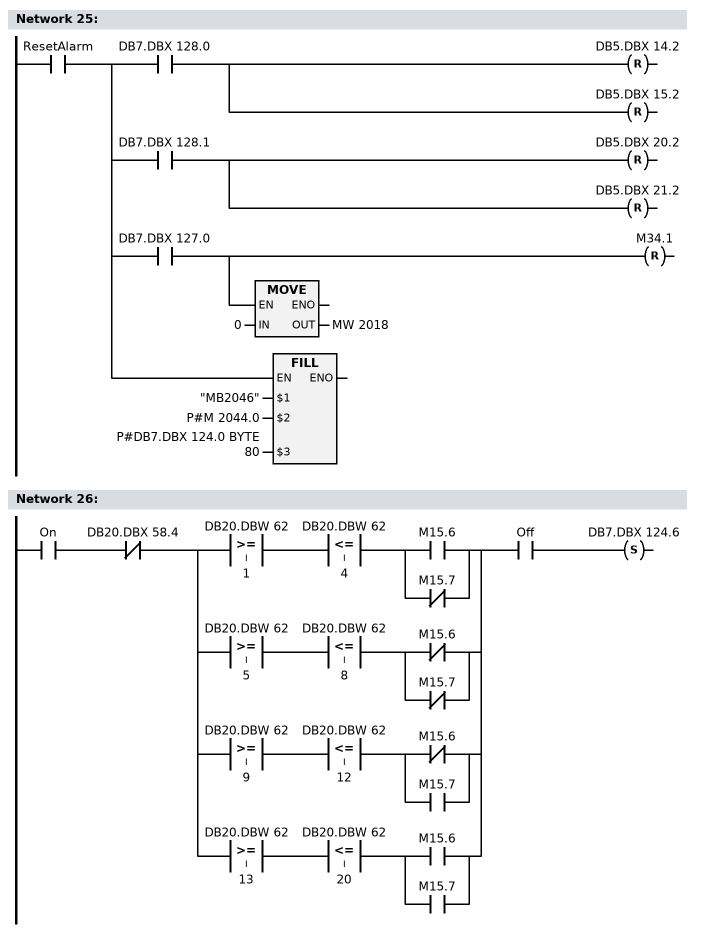
NETWORK
TITLE =
      A     "ResetAlarm";
      =     L 1.0;
      A     L 1.0;
      A     DB7.DBX 128.0;
      R     DB5.DBX 14.2;
      R     DB5.DBX 15.2;
      A     L 1.0;
      A     DB7.DBX 128.1;
      R     DB5.DBX 20.2;
      R     DB5.DBX 21.2;
      A     L 1.0;
      A     DB7.DBX 127.0;
      =     L 1.1;
      A     L 1.1;
      BLD   102;
      R     "M34.1";
      A     L 1.1;
      JNB   M001;
      L     0;
      T     MW 2018;
M001: NOP   0;
      A     L 1.0;
      JNB   M002;
      CALL  "FILL" (
           $1                       := "MB2046",
           $2                       := P#M 2044.0,
           $3                       := P#DB7.DBX 124.0 BYTE 80);
M002: NOP   0;
NETWORK
TITLE =
      A     "On";
      AN    DB20.DBX 58.4;
      A(;
      A(;
      L     DB20.DBW 62;
      L     1;
      >=I;
      );
      A(;
      L     DB20.DBW 62;
      L     4;
      <=I;
      );
      A(;
      O     "M15.6";
      ON    "M15.7";
      );
      O;
      A(;
      L     DB20.DBW 62;
      L     5;
      >=I;
      );
      A(;
      L     DB20.DBW 62;
      L     8;
      <=I;
      );
      A(;
      ON    "M15.6";
      ON    "M15.7";
      );
      O;
      A(;
      L     DB20.DBW 62;
      L     9;
      >=I;
      );
      A(;
      L     DB20.DBW 62;
      L     12;
      <=I;
      );
      A(;
      ON    "M15.6";
      O     "M15.7";
      );
      O;
      A(;
      L     DB20.DBW 62;
      L     13;
      >=I;
      );
      A(;
      L     DB20.DBW 62;
      L     20;
      <=I;
      );
      A(;
      O     "M15.6";
      O     "M15.7";
      );
      );
      A     "Off";
      S     DB7.DBX 124.6;
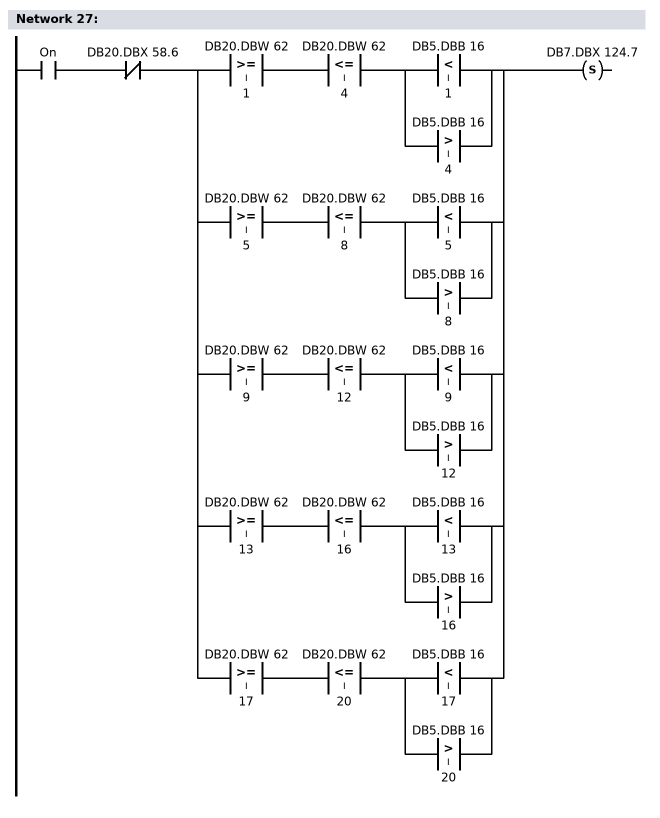
NETWORK
TITLE =
      A     "On";
      AN    DB20.DBX 58.6;
      A(;
      A(;
      L     DB20.DBW 62;
      L     1;
      >=I;
      );
      A(;
      L     DB20.DBW 62;
      L     4;
      <=I;
      );
      A(;
      O(;
      L     DB5.DBB 16;
      L     1;
      <I;
      );
      O(;
      L     DB5.DBB 16;
      L     4;
      >I;
      );
      );
      O;
      A(;
      L     DB20.DBW 62;
      L     5;
      >=I;
      );
      A(;
      L     DB20.DBW 62;
      L     8;
      <=I;
      );
      A(;
      O(;
      L     DB5.DBB 16;
      L     5;
      <I;
      );
      O(;
      L     DB5.DBB 16;
      L     8;
      >I;
      );
      );
      O;
      A(;
      L     DB20.DBW 62;
      L     9;
      >=I;
      );
      A(;
      L     DB20.DBW 62;
      L     12;
      <=I;
      );
      A(;
      O(;
      L     DB5.DBB 16;
      L     9;
      <I;
      );
      O(;
      L     DB5.DBB 16;
      L     12;
      >I;
      );
      );
      O;
      A(;
      L     DB20.DBW 62;
      L     13;
      >=I;
      );
      A(;
      L     DB20.DBW 62;
      L     16;
      <=I;
      );
      A(;
      O(;
      L     DB5.DBB 16;
      L     13;
      <I;
      );
      O(;
      L     DB5.DBB 16;
      L     16;
      >I;
      );
      );
      O;
      A(;
      L     DB20.DBW 62;
      L     17;
      >=I;
      );
      A(;
      L     DB20.DBW 62;
      L     20;
      <=I;
      );
      A(;
      O(;
      L     DB5.DBB 16;
      L     17;
      <I;
      );
      O(;
      L     DB5.DBB 16;
      L     20;
      >I;
      );
      );
      );
      S     DB7.DBX 124.7;
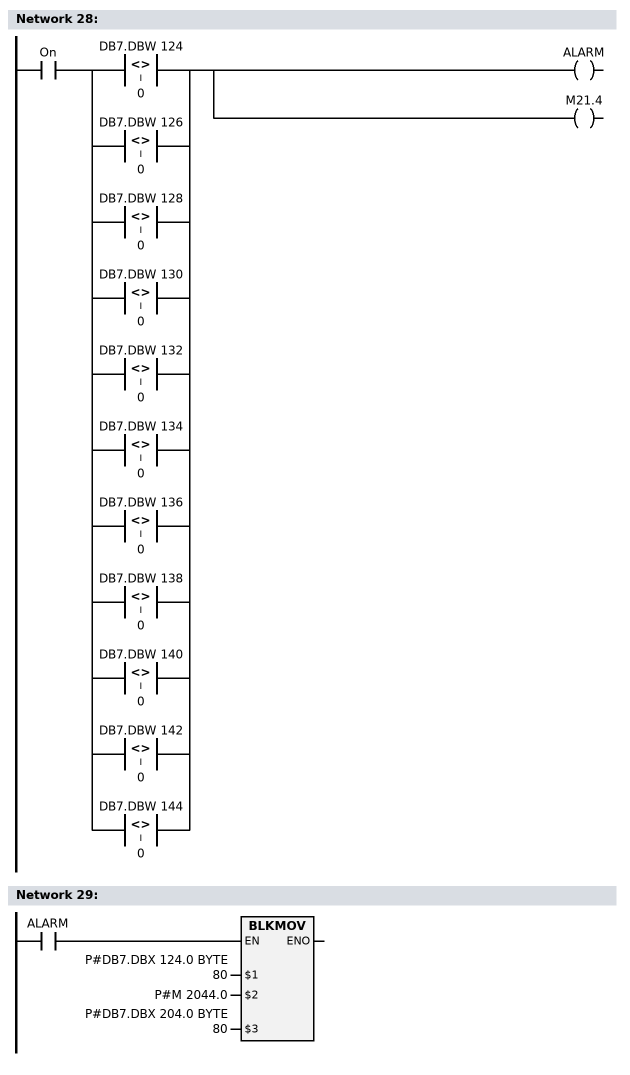
NETWORK
TITLE =
      A     "On";
      A(;
      O(;
      L     DB7.DBW 124;
      L     0;
      <>I;
      );
      O(;
      L     DB7.DBW 126;
      L     0;
      <>I;
      );
      O(;
      L     DB7.DBW 128;
      L     0;
      <>I;
      );
      O(;
      L     DB7.DBW 130;
      L     0;
      <>I;
      );
      O(;
      L     DB7.DBW 132;
      L     0;
      <>I;
      );
      O(;
      L     DB7.DBW 134;
      L     0;
      <>I;
      );
      O(;
      L     DB7.DBW 136;
      L     0;
      <>I;
      );
      O(;
      L     DB7.DBW 138;
      L     0;
      <>I;
      );
      O(;
      L     DB7.DBW 140;
      L     0;
      <>I;
      );
      O(;
      L     DB7.DBW 142;
      L     0;
      <>I;
      );
      O(;
      L     DB7.DBW 144;
      L     0;
      <>I;
      );
      );
      =     "ALARM";
      =     "M21.4";
NETWORK
TITLE =
      A     "ALARM";
      JNB   M003;
      CALL  "BLKMOV" (
           $1                       := P#DB7.DBX 124.0 BYTE 80,
           $2                       := P#M 2044.0,
           $3                       := P#DB7.DBX 204.0 BYTE 80);
M003: NOP   0;
END_FUNCTION

FUNCTION "FC17 - OPERATOR PANNEL" : VOID	// FC 17
VERSION : 0.1
BEGIN
// (block stored without names or comments; labels and parameter names are numbered)
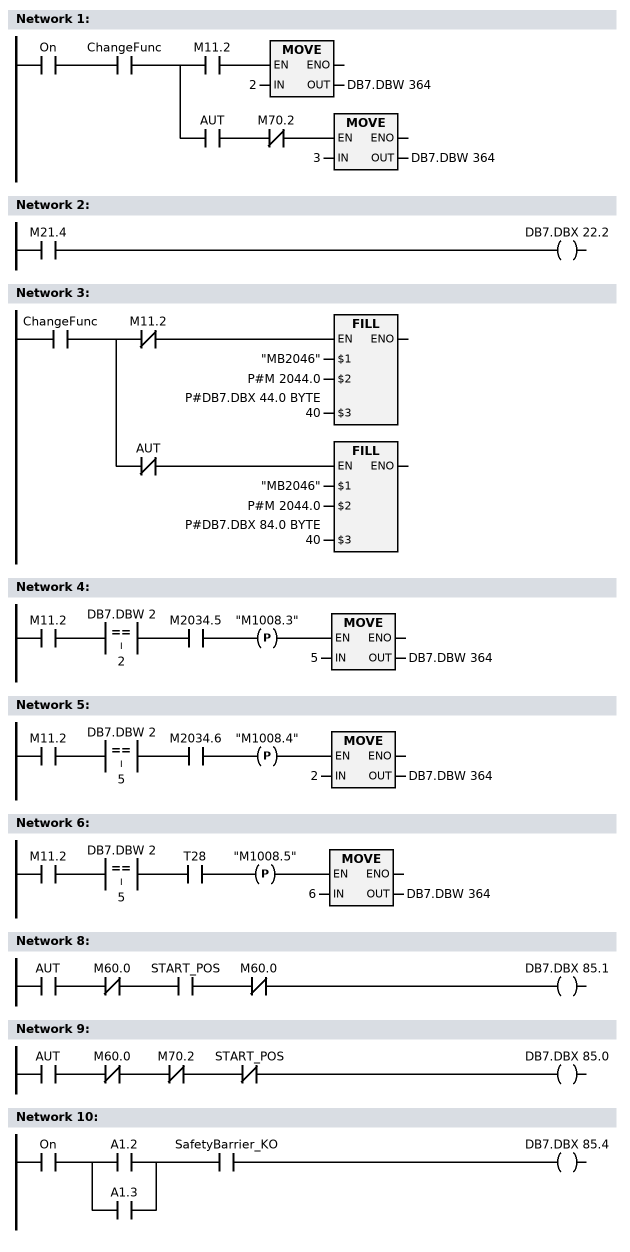
NETWORK
TITLE =
      A     "On";
      A     "ChangeFunc";
      =     L 0.0;
      A     L 0.0;
      A     "M11.2";
      JNB   M001;
      L     2;
      T     DB7.DBW 364;
M001: NOP   0;
      A     L 0.0;
      A     "AUT";
      AN    "M70.2";
      JNB   M002;
      L     3;
      T     DB7.DBW 364;
M002: NOP   0;
NETWORK
TITLE =
      A     "M21.4";
      =     DB7.DBX 22.2;
NETWORK
TITLE =
      A     "ChangeFunc";
      =     L 0.0;
      A     L 0.0;
      AN    "M11.2";
      JNB   M003;
      CALL  "FILL" (
           $1                       := "MB2046",
           $2                       := P#M 2044.0,
           $3                       := P#DB7.DBX 44.0 BYTE 40);
M003: NOP   0;
      A     L 0.0;
      AN    "AUT";
      JNB   M004;
      CALL  "FILL" (
           $1                       := "MB2046",
           $2                       := P#M 2044.0,
           $3                       := P#DB7.DBX 84.0 BYTE 40);
M004: NOP   0;
NETWORK
TITLE =
      A     "M11.2";
      A(;
      L     DB7.DBW 2;
      L     2;
      ==I;
      );
      A     "M2034.5";
      FP    "M1008.3";
      JNB   M005;
      L     5;
      T     DB7.DBW 364;
M005: NOP   0;
NETWORK
TITLE =
      A     "M11.2";
      A(;
      L     DB7.DBW 2;
      L     5;
      ==I;
      );
      A     "M2034.6";
      FP    "M1008.4";
      JNB   M006;
      L     2;
      T     DB7.DBW 364;
M006: NOP   0;
NETWORK
TITLE =
      A     "M11.2";
      A(;
      L     DB7.DBW 2;
      L     5;
      ==I;
      );
      A     "T28";
      FP    "M1008.5";
      JNB   M007;
      L     6;
      T     DB7.DBW 364;
M007: NOP   0;
NETWORK
TITLE =
NETWORK
TITLE =
      A     "AUT";
      AN    "M60.0";
      A     "START_POS";
      AN    "M60.0";
      =     DB7.DBX 85.1;
NETWORK
TITLE =
      A     "AUT";
      AN    "M60.0";
      AN    "M70.2";
      AN    "START_POS";
      =     DB7.DBX 85.0;
NETWORK
TITLE =
      A     "On";
      A(;
      O     "A1.2";
      O     "A1.3";
      );
      A     "SafetyBarrier_KO";
      =     DB7.DBX 85.4;
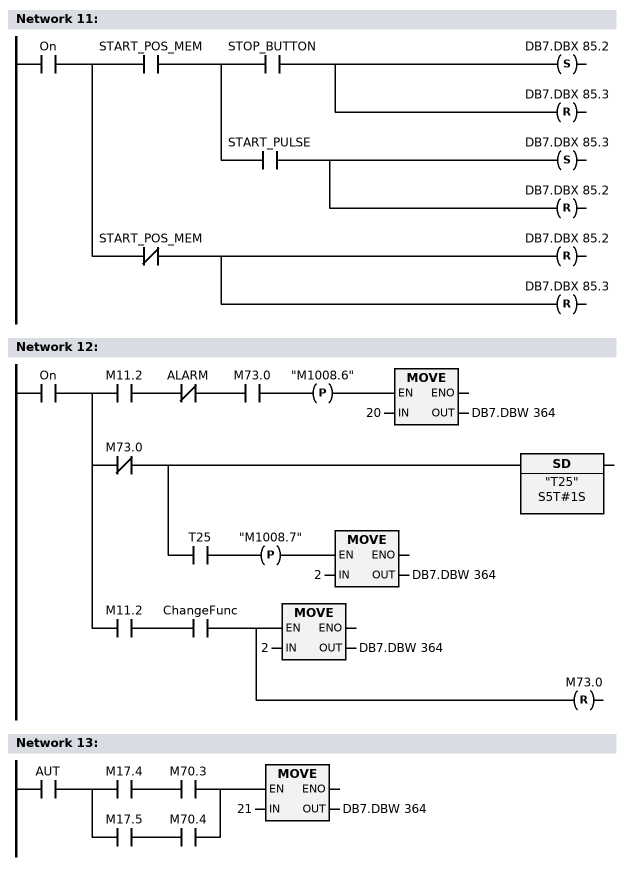
NETWORK
TITLE =
      A     "On";
      =     L 0.0;
      A     L 0.0;
      A     "START_POS_MEM";
      =     L 0.1;
      A     L 0.1;
      A     "STOP_BUTTON";
      S     DB7.DBX 85.2;
      R     DB7.DBX 85.3;
      A     L 0.1;
      A     "START_PULSE";
      S     DB7.DBX 85.3;
      R     DB7.DBX 85.2;
      A     L 0.0;
      AN    "START_POS_MEM";
      R     DB7.DBX 85.2;
      R     DB7.DBX 85.3;
NETWORK
TITLE =
      A     "On";
      =     L 0.0;
      A     L 0.0;
      A     "M11.2";
      AN    "ALARM";
      A     "M73.0";
      FP    "M1008.6";
      JNB   M008;
      L     20;
      T     DB7.DBW 364;
M008: NOP   0;
      A     L 0.0;
      AN    "M73.0";
      =     L 0.1;
      A     L 0.1;
      BLD   102;
      L     S5T#1S;
      SD    "T25";
      A     L 0.1;
      A     "T25";
      FP    "M1008.7";
      JNB   M009;
      L     2;
      T     DB7.DBW 364;
M009: NOP   0;
      A     L 0.0;
      A     "M11.2";
      A     "ChangeFunc";
      =     L 0.1;
      A     L 0.1;
      JNB   M010;
      L     2;
      T     DB7.DBW 364;
M010: NOP   0;
      A     L 0.1;
      BLD   102;
      R     "M73.0";
NETWORK
TITLE =
      A     "AUT";
      A(;
      A     "M17.4";
      A     "M70.3";
      O;
      A     "M17.5";
      A     "M70.4";
      );
      JNB   M011;
      L     21;
      T     DB7.DBW 364;
M011: NOP   0;
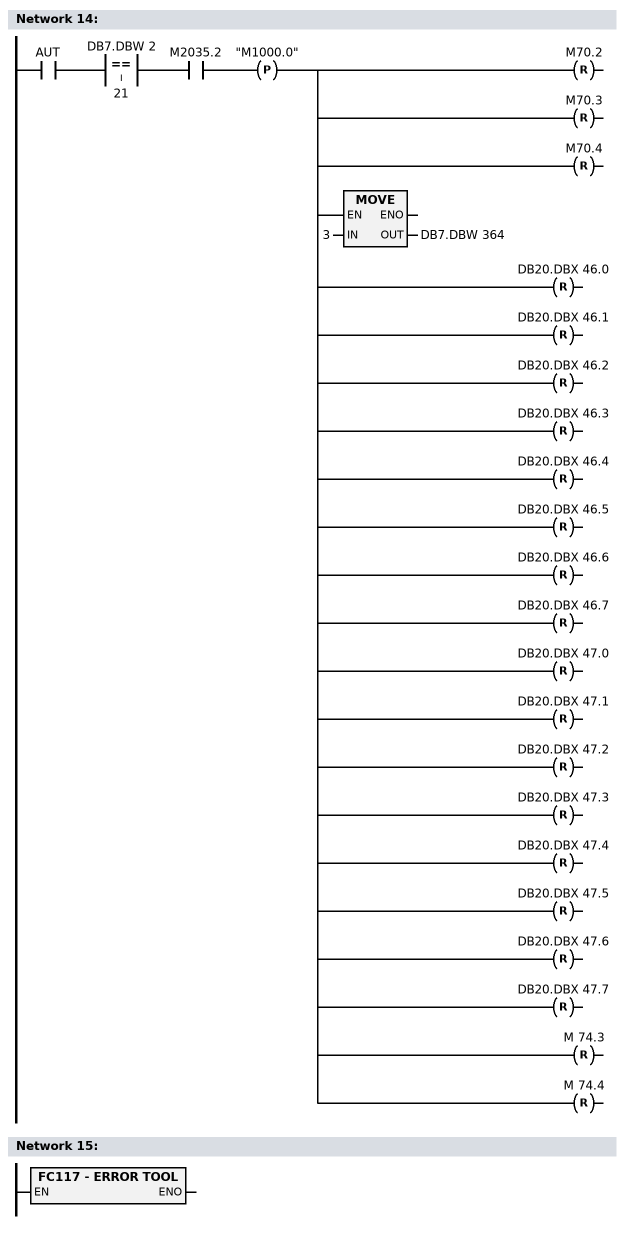
NETWORK
TITLE =
      A     "AUT";
      A(;
      L     DB7.DBW 2;
      L     21;
      ==I;
      );
      A     "M2035.2";
      FP    "M1000.0";
      =     L 0.0;
      A     L 0.0;
      BLD   102;
      R     "M70.2";
      A     L 0.0;
      BLD   102;
      R     "M70.3";
      A     L 0.0;
      BLD   102;
      R     "M70.4";
      A     L 0.0;
      JNB   M012;
      L     3;
      T     DB7.DBW 364;
M012: NOP   0;
      A     L 0.0;
      BLD   102;
      R     DB20.DBX 46.0;
      A     L 0.0;
      BLD   102;
      R     DB20.DBX 46.1;
      A     L 0.0;
      BLD   102;
      R     DB20.DBX 46.2;
      A     L 0.0;
      BLD   102;
      R     DB20.DBX 46.3;
      A     L 0.0;
      BLD   102;
      R     DB20.DBX 46.4;
      A     L 0.0;
      BLD   102;
      R     DB20.DBX 46.5;
      A     L 0.0;
      BLD   102;
      R     DB20.DBX 46.6;
      A     L 0.0;
      BLD   102;
      R     DB20.DBX 46.7;
      A     L 0.0;
      BLD   102;
      R     DB20.DBX 47.0;
      A     L 0.0;
      BLD   102;
      R     DB20.DBX 47.1;
      A     L 0.0;
      BLD   102;
      R     DB20.DBX 47.2;
      A     L 0.0;
      BLD   102;
      R     DB20.DBX 47.3;
      A     L 0.0;
      BLD   102;
      R     DB20.DBX 47.4;
      A     L 0.0;
      BLD   102;
      R     DB20.DBX 47.5;
      A     L 0.0;
      BLD   102;
      R     DB20.DBX 47.6;
      A     L 0.0;
      BLD   102;
      R     DB20.DBX 47.7;
      A     L 0.0;
      BLD   102;
      R     M 74.3;
      A     L 0.0;
      BLD   102;
      R     M 74.4;
NETWORK
TITLE =
      CALL  "FC117 - ERROR TOOL";
      NOP   0;
END_FUNCTION

FUNCTION "FC18 - OUTPUTS" : VOID	// FC 18
VERSION : 0.1
BEGIN
// (block stored without names or comments; labels and parameter names are numbered)
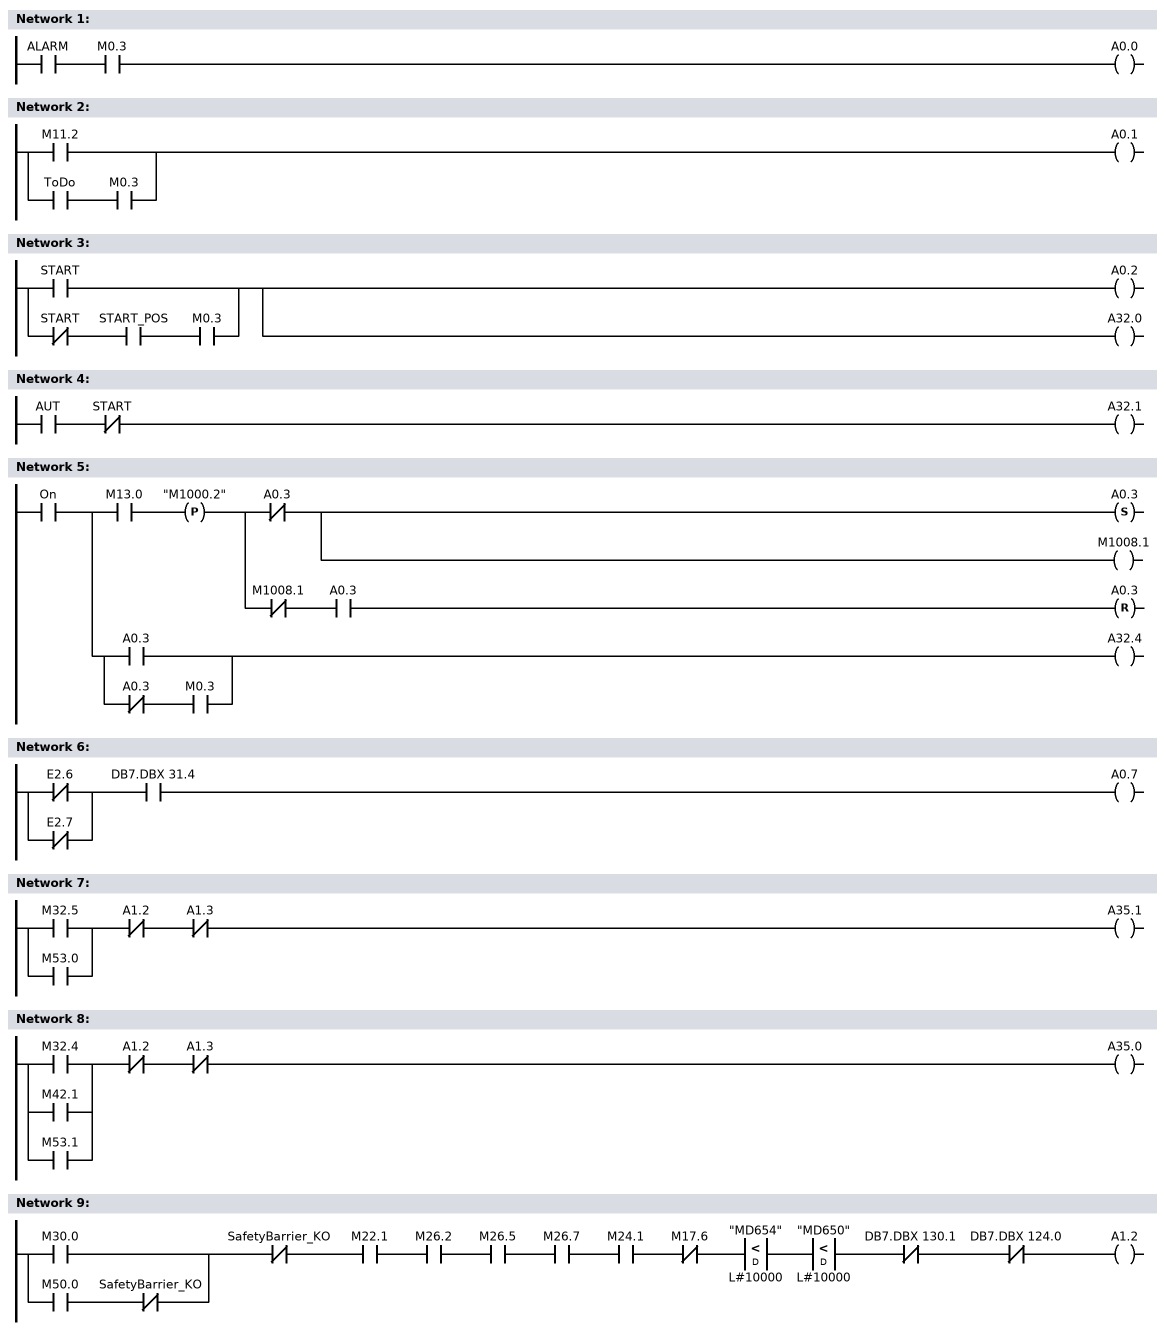
NETWORK
TITLE =
      A     "ALARM";
      A     "M0.3";
      =     "A0.0";
NETWORK
TITLE =
      O     "M11.2";
      O;
      A     "ToDo";
      A     "M0.3";
      =     "A0.1";
NETWORK
TITLE =
      O     "START";
      O;
      AN    "START";
      A     "START_POS";
      A     "M0.3";
      =     "A0.2";
      =     "A32.0";
NETWORK
TITLE =
      A     "AUT";
      AN    "START";
      =     "A32.1";
NETWORK
TITLE =
      A     "On";
      =     L 0.0;
      A     L 0.0;
      A     "M13.0";
      FP    "M1000.2";
      =     L 0.1;
      A     L 0.1;
      AN    "A0.3";
      S     "A0.3";
      =     "M1008.1";
      A     L 0.1;
      AN    "M1008.1";
      A     "A0.3";
      R     "A0.3";
      A     L 0.0;
      A(;
      O     "A0.3";
      O;
      AN    "A0.3";
      A     "M0.3";
      );
      =     "A32.4";
NETWORK
TITLE =
      A(;
      ON    "E2.6";
      ON    "E2.7";
      );
      A     DB7.DBX 31.4;
      =     "A0.7";
NETWORK
TITLE =
      A(;
      O     "M32.5";
      O     "M53.0";
      );
      AN    "A1.2";
      AN    "A1.3";
      =     "A35.1";
NETWORK
TITLE =
      A(;
      O     "M32.4";
      O     "M42.1";
      O     "M53.1";
      );
      AN    "A1.2";
      AN    "A1.3";
      =     "A35.0";
NETWORK
TITLE =
      A(;
      O     "M30.0";
      O;
      A     "M50.0";
      AN    "SafetyBarrier_KO";
      );
      AN    "SafetyBarrier_KO";
      A     "M22.1";
      A     "M26.2";
      A     "M26.5";
      A     "M26.7";
      A     "M24.1";
      AN    "M17.6";
      A(;
      L     "MD654";
      L     L#10000;
      <D;
      );
      A(;
      L     "MD650";
      L     L#10000;
      <D;
      );
      AN    DB7.DBX 130.1;
      AN    DB7.DBX 124.0;
      =     "A1.2";
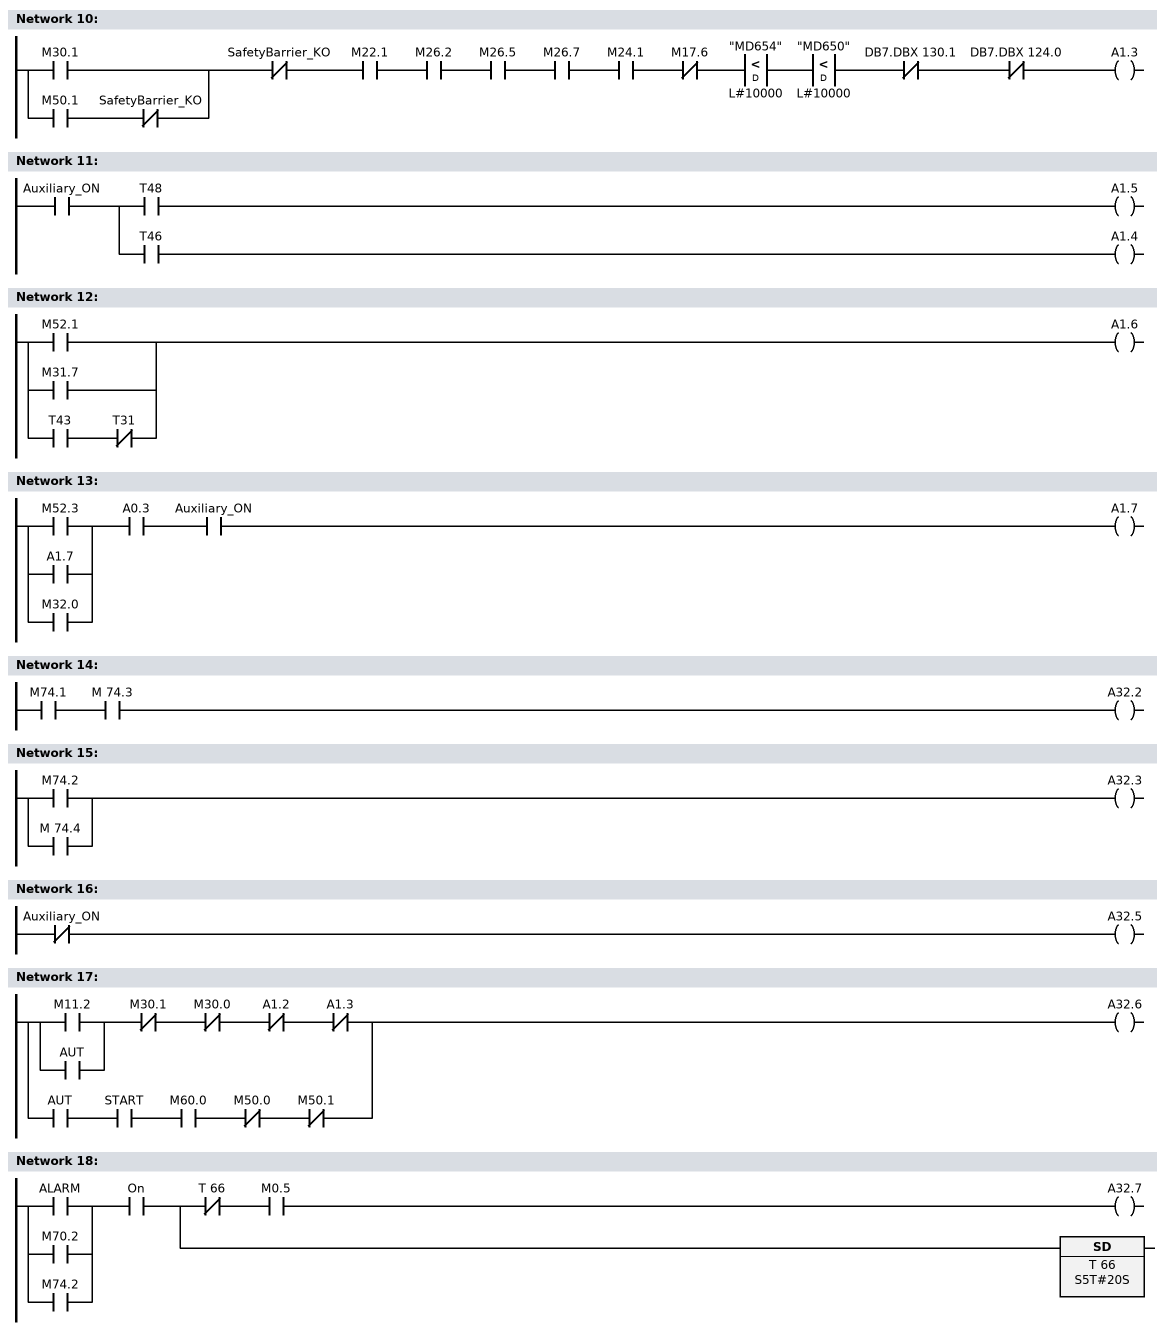
NETWORK
TITLE =
      A(;
      O     "M30.1";
      O;
      A     "M50.1";
      AN    "SafetyBarrier_KO";
      );
      AN    "SafetyBarrier_KO";
      A     "M22.1";
      A     "M26.2";
      A     "M26.5";
      A     "M26.7";
      A     "M24.1";
      AN    "M17.6";
      A(;
      L     "MD654";
      L     L#10000;
      <D;
      );
      A(;
      L     "MD650";
      L     L#10000;
      <D;
      );
      AN    DB7.DBX 130.1;
      AN    DB7.DBX 124.0;
      =     "A1.3";
NETWORK
TITLE =
      A     "Auxiliary_ON";
      =     L 0.0;
      A     L 0.0;
      A     "T48";
      =     "A1.5";
      A     L 0.0;
      A     "T46";
      =     "A1.4";
NETWORK
TITLE =
      O     "M52.1";
      O     "M31.7";
      O;
      A     "T43";
      AN    "T31";
      =     "A1.6";
NETWORK
TITLE =
      A(;
      O     "M52.3";
      O     "A1.7";
      O     "M32.0";
      );
      A     "A0.3";
      A     "Auxiliary_ON";
      =     "A1.7";
NETWORK
TITLE =
      A     "M74.1";
      A     M 74.3;
      =     "A32.2";
NETWORK
TITLE =
      O     "M74.2";
      O     M 74.4;
      =     "A32.3";
NETWORK
TITLE =
      AN    "Auxiliary_ON";
      =     "A32.5";
NETWORK
TITLE =
      A(;
      O     "M11.2";
      O     "AUT";
      );
      AN    "M30.1";
      AN    "M30.0";
      AN    "A1.2";
      AN    "A1.3";
      O;
      A     "AUT";
      A     "START";
      A     "M60.0";
      AN    "M50.0";
      AN    "M50.1";
      =     "A32.6";
NETWORK
TITLE =
      A(;
      O     "ALARM";
      O     "M70.2";
      O     "M74.2";
      );
      A     "On";
      =     L 0.0;
      A     L 0.0;
      AN    T 66;
      A     "M0.5";
      =     "A32.7";
      A     L 0.0;
      BLD   102;
      L     S5T#20S;
      SD    T 66;
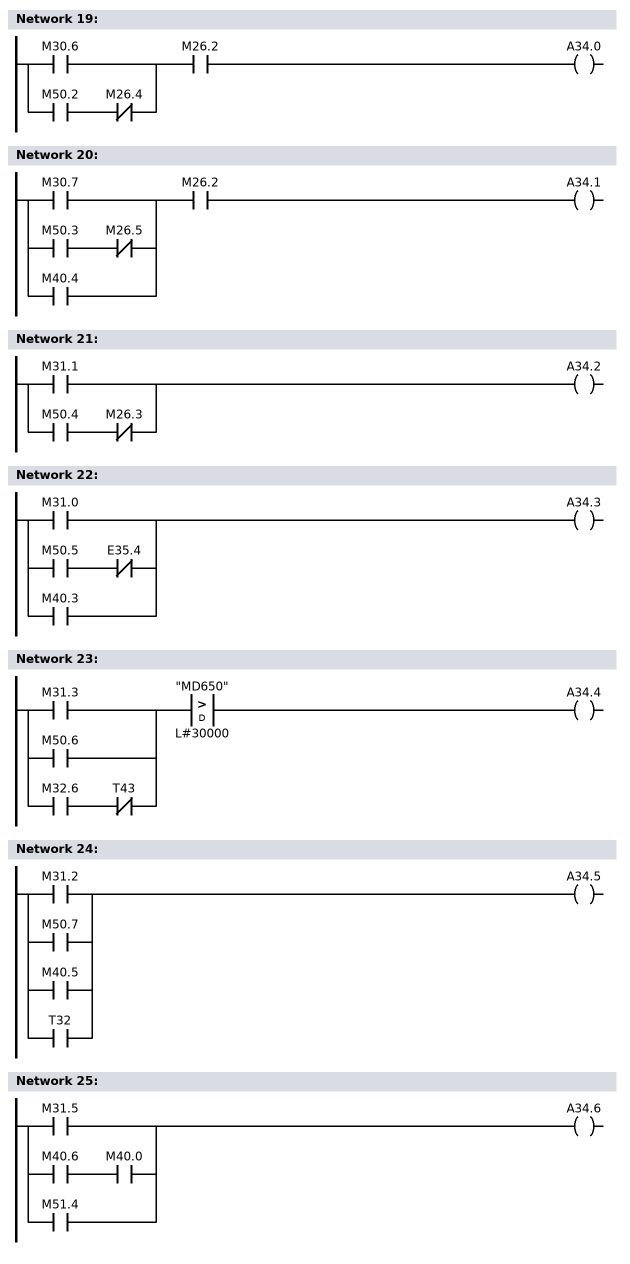
NETWORK
TITLE =
      A(;
      O     "M30.6";
      O;
      A     "M50.2";
      AN    "M26.4";
      );
      A     "M26.2";
      =     "A34.0";
NETWORK
TITLE =
      A(;
      O     "M30.7";
      O;
      A     "M50.3";
      AN    "M26.5";
      O     "M40.4";
      );
      A     "M26.2";
      =     "A34.1";
NETWORK
TITLE =
      O     "M31.1";
      O;
      A     "M50.4";
      AN    "M26.3";
      =     "A34.2";
NETWORK
TITLE =
      O     "M31.0";
      O;
      A     "M50.5";
      AN    "E35.4";
      O     "M40.3";
      =     "A34.3";
NETWORK
TITLE =
      A(;
      O     "M31.3";
      O     "M50.6";
      O;
      A     "M32.6";
      AN    "T43";
      );
      A(;
      L     "MD650";
      L     L#30000;
      >D;
      );
      =     "A34.4";
NETWORK
TITLE =
      O     "M31.2";
      O     "M50.7";
      O     "M40.5";
      O     "T32";
      =     "A34.5";
NETWORK
TITLE =
      O     "M31.5";
      O;
      A     "M40.6";
      A     "M40.0";
      O     "M51.4";
      =     "A34.6";
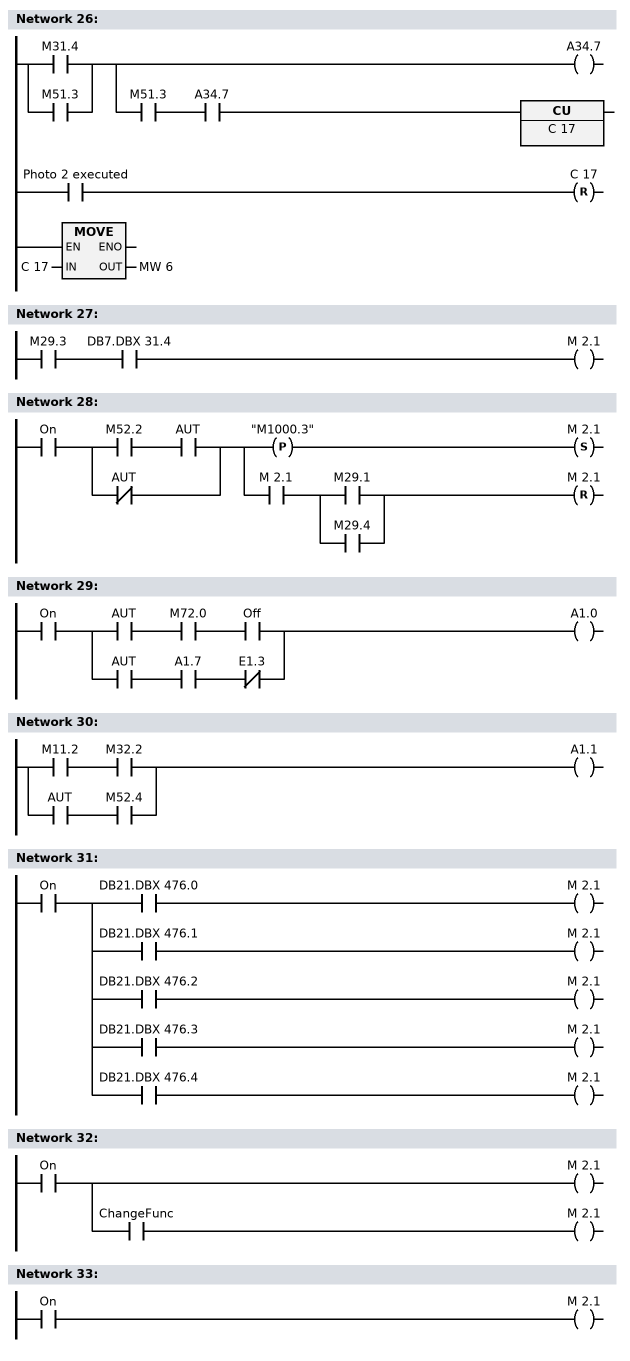
NETWORK
TITLE =
      O     "M31.4";
      O     "M51.3";
      =     L 0.0;
      A     L 0.0;
      BLD   102;
      =     "A34.7";
      A     L 0.0;
      A     "M51.3";
      A     "A34.7";
      CU    C 17;
      BLD   101;
      NOP   0;
      NOP   0;
      A     "Photo 2 executed";
      R     C 17;
      L     C 17;
      T     MW 6;
      NOP   0;
      NOP   0;
NETWORK
TITLE =
      A     "M29.3";
      A     DB7.DBX 31.4;
      =     M 2.1;
NETWORK
TITLE =
      A     "On";
      A(;
      A     "M52.2";
      A     "AUT";
      ON    "AUT";
      );
      =     L 0.0;
      A     L 0.0;
      FP    "M1000.3";
      S     M 2.1;
      A     L 0.0;
      A     M 2.1;
      A(;
      O     "M29.1";
      O     "M29.4";
      );
      R     M 2.1;
NETWORK
TITLE =
      A     "On";
      A(;
      A     "AUT";
      A     "M72.0";
      A     "Off";
      O;
      A     "AUT";
      A     "A1.7";
      AN    "E1.3";
      );
      =     "A1.0";
NETWORK
TITLE =
      A     "M11.2";
      A     "M32.2";
      O;
      A     "AUT";
      A     "M52.4";
      =     "A1.1";
NETWORK
TITLE =
      A     "On";
      =     L 0.0;
      A     L 0.0;
      A     DB21.DBX 476.0;
      =     M 2.1;
      A     L 0.0;
      A     DB21.DBX 476.1;
      =     M 2.1;
      A     L 0.0;
      A     DB21.DBX 476.2;
      =     M 2.1;
      A     L 0.0;
      A     DB21.DBX 476.3;
      =     M 2.1;
      A     L 0.0;
      A     DB21.DBX 476.4;
      =     M 2.1;
NETWORK
TITLE =
      A     "On";
      =     L 0.0;
      A     L 0.0;
      BLD   102;
      =     M 2.1;
      A     L 0.0;
      A     "ChangeFunc";
      =     M 2.1;
NETWORK
TITLE =
      A     "On";
      =     M 2.1;
END_FUNCTION

FUNCTION "FC19 - REPOSITIONING" : VOID	// FC 19
VERSION : 0.1
BEGIN
// (block stored without names or comments; labels and parameter names are numbered)
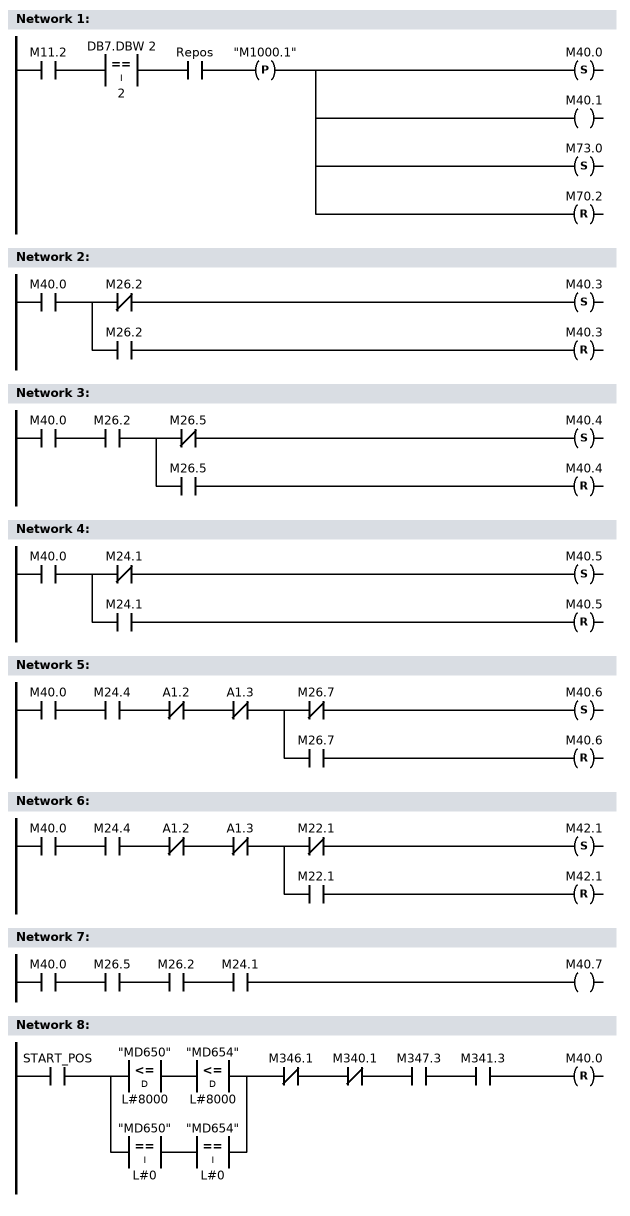
NETWORK
TITLE =
      A     "M11.2";
      A(;
      L     DB7.DBW 2;
      L     2;
      ==I;
      );
      A     "Repos";
      FP    "M1000.1";
      S     "M40.0";
      =     "M40.1";
      S     "M73.0";
      R     "M70.2";
NETWORK
TITLE =
      A     "M40.0";
      =     L 0.0;
      A     L 0.0;
      AN    "M26.2";
      S     "M40.3";
      A     L 0.0;
      A     "M26.2";
      R     "M40.3";
NETWORK
TITLE =
      A     "M40.0";
      A     "M26.2";
      =     L 0.0;
      A     L 0.0;
      AN    "M26.5";
      S     "M40.4";
      A     L 0.0;
      A     "M26.5";
      R     "M40.4";
NETWORK
TITLE =
      A     "M40.0";
      =     L 0.0;
      A     L 0.0;
      AN    "M24.1";
      S     "M40.5";
      A     L 0.0;
      A     "M24.1";
      R     "M40.5";
NETWORK
TITLE =
      A     "M40.0";
      A     "M24.4";
      AN    "A1.2";
      AN    "A1.3";
      =     L 0.0;
      A     L 0.0;
      AN    "M26.7";
      S     "M40.6";
      A     L 0.0;
      A     "M26.7";
      R     "M40.6";
NETWORK
TITLE =
      A     "M40.0";
      A     "M24.4";
      AN    "A1.2";
      AN    "A1.3";
      =     L 0.0;
      A     L 0.0;
      AN    "M22.1";
      S     "M42.1";
      A     L 0.0;
      A     "M22.1";
      R     "M42.1";
NETWORK
TITLE =
      A     "M40.0";
      A     "M26.5";
      A     "M26.2";
      A     "M24.1";
      =     "M40.7";
NETWORK
TITLE =
      A     "START_POS";
      A(;
      A(;
      L     "MD650";
      L     L#8000;
      <=D;
      );
      A(;
      L     "MD654";
      L     L#8000;
      <=D;
      );
      O;
      A(;
      L     "MD650";
      L     L#0;
      ==I;
      );
      A(;
      L     "MD654";
      L     L#0;
      ==I;
      );
      );
      AN    "M346.1";
      AN    "M340.1";
      A     "M347.3";
      A     "M341.3";
      R     "M40.0";
NETWORK
TITLE =
END_FUNCTION

FUNCTION "FC - AUTOMATIC" : VOID	// FC 24
VERSION : 0.1
BEGIN
// (block stored without names or comments; labels and parameter names are numbered)
